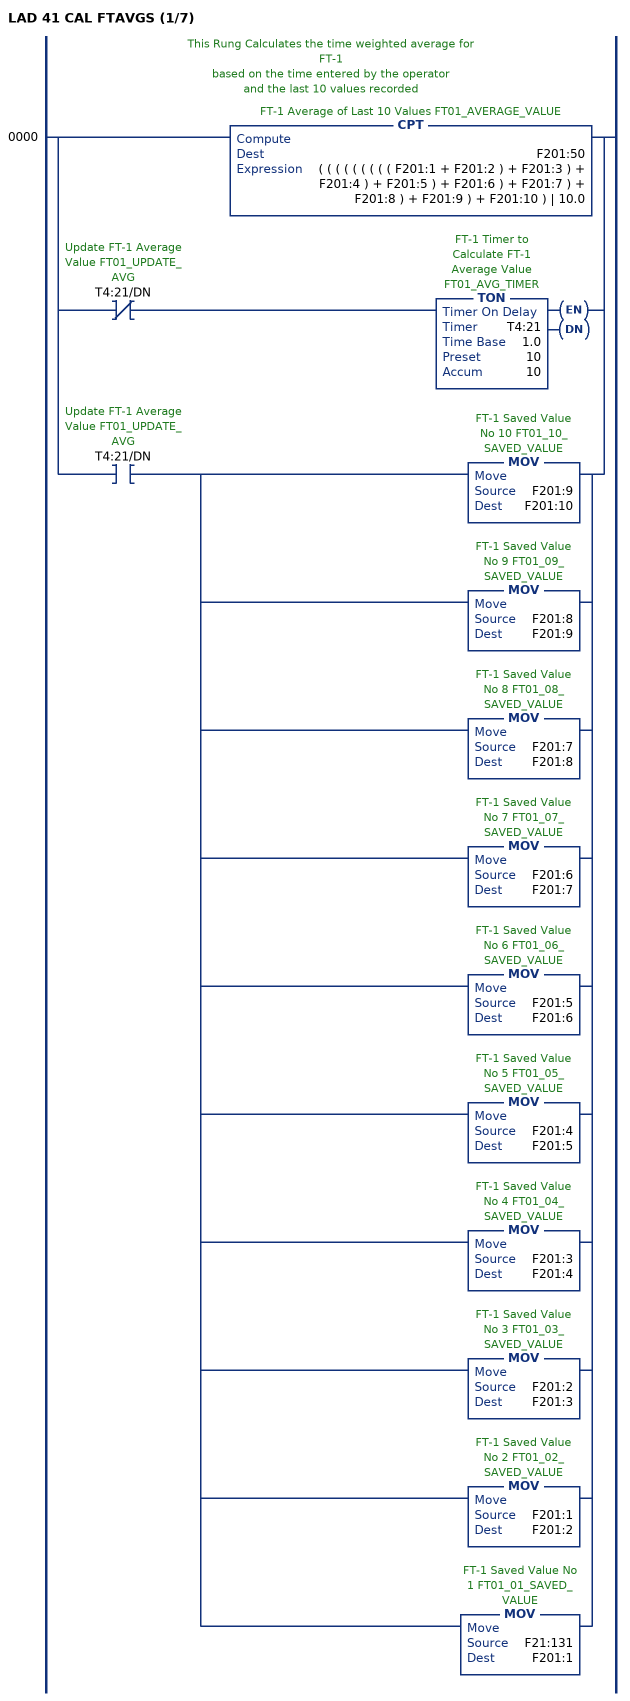
% Rung: 0 %
% This Rung Calculates the time weighted average for
% FT-1
% based on the time entered by the operator
% and the last 10 values recorded %
SOR BST CPT F201:50 " ( ( ( ( ( ( ( ( ( F201:1 + F201:2 ) + F201:3 ) + F201:4 ) + F201:5 ) + F201:6 ) + F201:7 ) + F201:8 ) + F201:9 ) + F201:10 ) | 10.0 " NXB XIO T4:21/DN TON T4:21 1.0 10 10 NXB XIC T4:21/DN BST MOV F201:9 F201:10 NXB MOV F201:8 F201:9 NXB MOV F201:7 F201:8 NXB MOV F201:6 F201:7 NXB MOV F201:5 F201:6 NXB MOV F201:4 F201:5 NXB MOV F201:3 F201:4 NXB MOV F201:2 F201:3 NXB MOV F201:1 F201:2 NXB MOV F21:131 F201:1 BND BND EOR
%   F201:50  FT01_AVERAGE_VALUE  "FT-1 Average of Last 10 Values" %
%   F201:1  FT01_01_SAVED_VALUE  "FT-1 Saved Value No 1" %
%   F201:2  FT01_02_SAVED_VALUE  "FT-1 Saved Value No 2" %
%   F201:3  FT01_03_SAVED_VALUE  "FT-1 Saved Value No 3" %
%   F201:4  FT01_04_SAVED_VALUE  "FT-1 Saved Value No 4" %
%   F201:5  FT01_05_SAVED_VALUE  "FT-1 Saved Value No 5" %
%   F201:6  FT01_06_SAVED_VALUE  "FT-1 Saved Value No 6" %
%   F201:7  FT01_07_SAVED_VALUE  "FT-1 Saved Value No 7" %
%   F201:8  FT01_08_SAVED_VALUE  "FT-1 Saved Value No 8" %
%   F201:9  FT01_09_SAVED_VALUE  "FT-1 Saved Value No 9" %
%   F201:10  FT01_10_SAVED_VALUE  "FT-1 Saved Value No 10" %
%   T4:21/DN  FT01_UPDATE_AVG  "Update FT-1 Average Value" %
%   T4:21  FT01_AVG_TIMER  "FT-1 Timer to Calculate FT-1 Average Value" %
%   F21:131  FT01  "FT-1 Flow Transmitter No-1" %

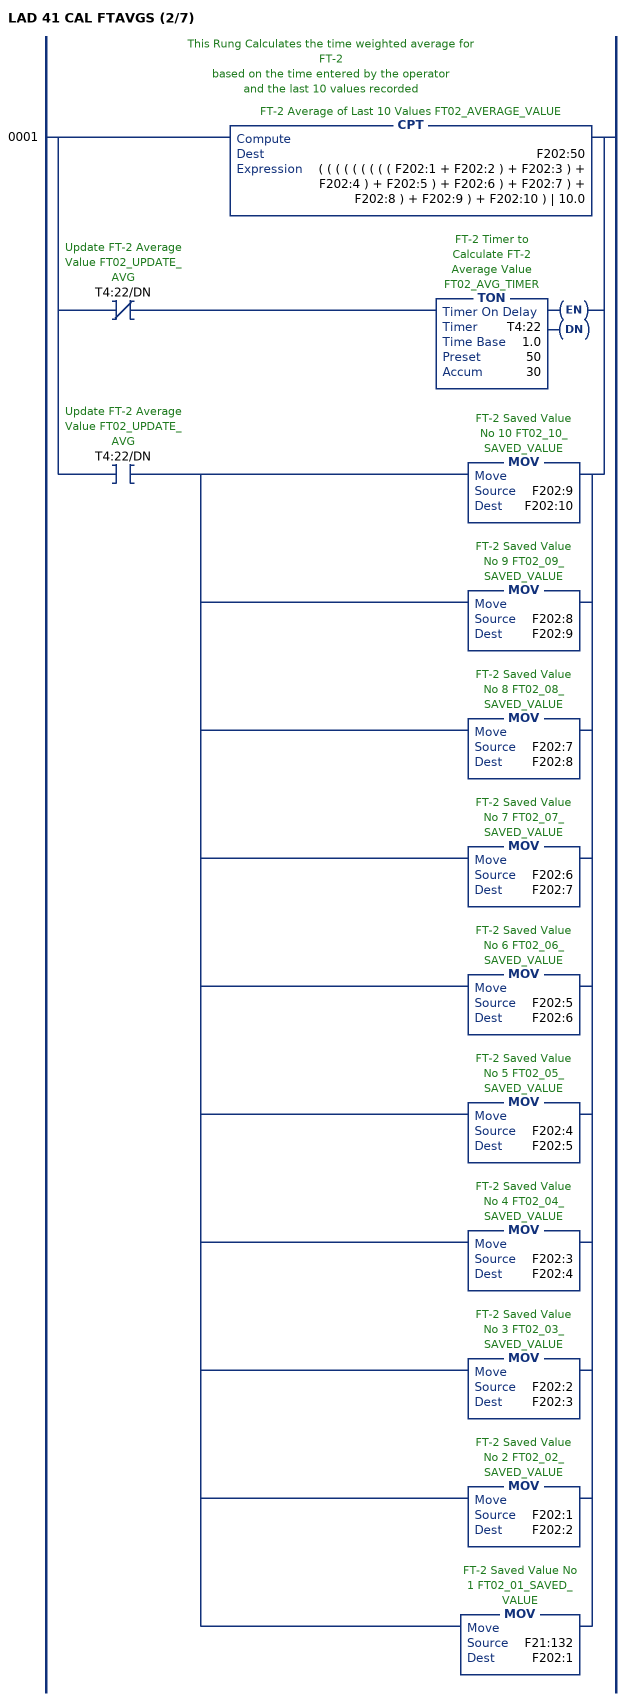
% Rung: 1 %
% This Rung Calculates the time weighted average for
% FT-2
% based on the time entered by the operator
% and the last 10 values recorded %
SOR BST CPT F202:50 " ( ( ( ( ( ( ( ( ( F202:1 + F202:2 ) + F202:3 ) + F202:4 ) + F202:5 ) + F202:6 ) + F202:7 ) + F202:8 ) + F202:9 ) + F202:10 ) | 10.0 " NXB XIO T4:22/DN TON T4:22 1.0 50 30 NXB XIC T4:22/DN BST MOV F202:9 F202:10 NXB MOV F202:8 F202:9 NXB MOV F202:7 F202:8 NXB MOV F202:6 F202:7 NXB MOV F202:5 F202:6 NXB MOV F202:4 F202:5 NXB MOV F202:3 F202:4 NXB MOV F202:2 F202:3 NXB MOV F202:1 F202:2 NXB MOV F21:132 F202:1 BND BND EOR
%   F202:50  FT02_AVERAGE_VALUE  "FT-2 Average of Last 10 Values" %
%   F202:1  FT02_01_SAVED_VALUE  "FT-2 Saved Value No 1" %
%   F202:2  FT02_02_SAVED_VALUE  "FT-2 Saved Value No 2" %
%   F202:3  FT02_03_SAVED_VALUE  "FT-2 Saved Value No 3" %
%   F202:4  FT02_04_SAVED_VALUE  "FT-2 Saved Value No 4" %
%   F202:5  FT02_05_SAVED_VALUE  "FT-2 Saved Value No 5" %
%   F202:6  FT02_06_SAVED_VALUE  "FT-2 Saved Value No 6" %
%   F202:7  FT02_07_SAVED_VALUE  "FT-2 Saved Value No 7" %
%   F202:8  FT02_08_SAVED_VALUE  "FT-2 Saved Value No 8" %
%   F202:9  FT02_09_SAVED_VALUE  "FT-2 Saved Value No 9" %
%   F202:10  FT02_10_SAVED_VALUE  "FT-2 Saved Value No 10" %
%   T4:22/DN  FT02_UPDATE_AVG  "Update FT-2 Average Value" %
%   T4:22  FT02_AVG_TIMER  "FT-2 Timer to Calculate FT-2 Average Value" %
%   F21:132  FT02  "FT-2 Flow Transmitter No-2" %

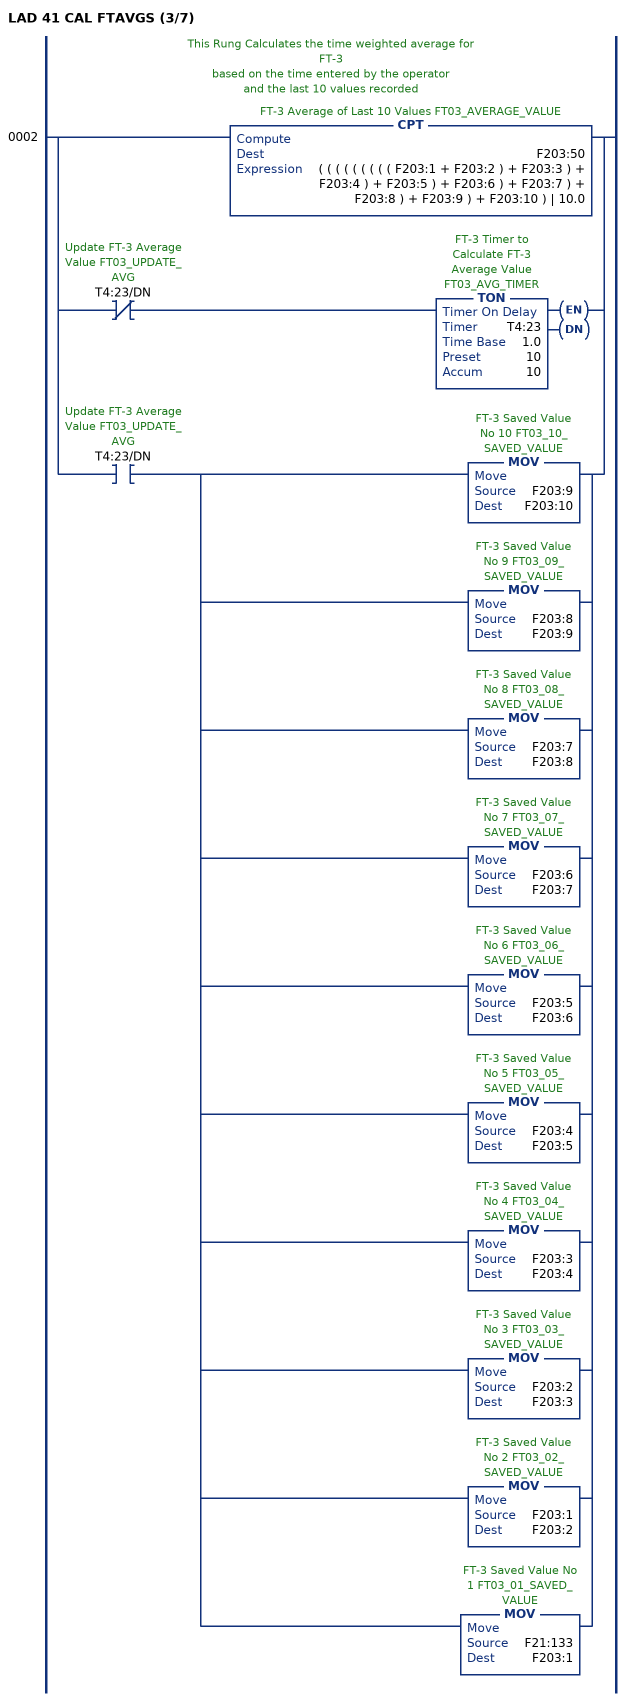
% Rung: 2 %
% This Rung Calculates the time weighted average for
% FT-3
% based on the time entered by the operator
% and the last 10 values recorded %
SOR BST CPT F203:50 " ( ( ( ( ( ( ( ( ( F203:1 + F203:2 ) + F203:3 ) + F203:4 ) + F203:5 ) + F203:6 ) + F203:7 ) + F203:8 ) + F203:9 ) + F203:10 ) | 10.0 " NXB XIO T4:23/DN TON T4:23 1.0 10 10 NXB XIC T4:23/DN BST MOV F203:9 F203:10 NXB MOV F203:8 F203:9 NXB MOV F203:7 F203:8 NXB MOV F203:6 F203:7 NXB MOV F203:5 F203:6 NXB MOV F203:4 F203:5 NXB MOV F203:3 F203:4 NXB MOV F203:2 F203:3 NXB MOV F203:1 F203:2 NXB MOV F21:133 F203:1 BND BND EOR
%   F203:50  FT03_AVERAGE_VALUE  "FT-3 Average of Last 10 Values" %
%   F203:1  FT03_01_SAVED_VALUE  "FT-3 Saved Value No 1" %
%   F203:2  FT03_02_SAVED_VALUE  "FT-3 Saved Value No 2" %
%   F203:3  FT03_03_SAVED_VALUE  "FT-3 Saved Value No 3" %
%   F203:4  FT03_04_SAVED_VALUE  "FT-3 Saved Value No 4" %
%   F203:5  FT03_05_SAVED_VALUE  "FT-3 Saved Value No 5" %
%   F203:6  FT03_06_SAVED_VALUE  "FT-3 Saved Value No 6" %
%   F203:7  FT03_07_SAVED_VALUE  "FT-3 Saved Value No 7" %
%   F203:8  FT03_08_SAVED_VALUE  "FT-3 Saved Value No 8" %
%   F203:9  FT03_09_SAVED_VALUE  "FT-3 Saved Value No 9" %
%   F203:10  FT03_10_SAVED_VALUE  "FT-3 Saved Value No 10" %
%   T4:23/DN  FT03_UPDATE_AVG  "Update FT-3 Average Value" %
%   T4:23  FT03_AVG_TIMER  "FT-3 Timer to Calculate FT-3 Average Value" %
%   F21:133  FT03  "FT-3 Flow Transmitter No-3" %

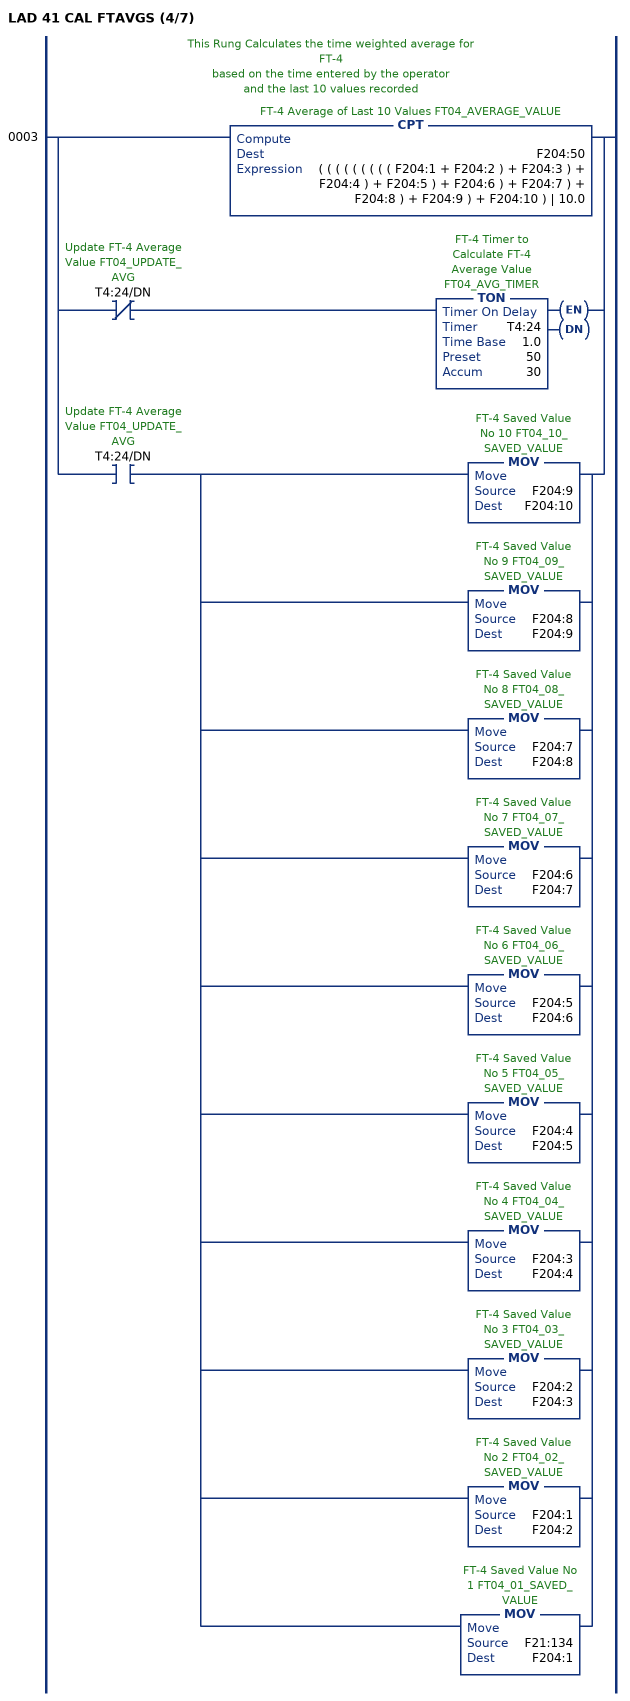
% Rung: 3 %
% This Rung Calculates the time weighted average for
% FT-4
% based on the time entered by the operator
% and the last 10 values recorded %
SOR BST CPT F204:50 " ( ( ( ( ( ( ( ( ( F204:1 + F204:2 ) + F204:3 ) + F204:4 ) + F204:5 ) + F204:6 ) + F204:7 ) + F204:8 ) + F204:9 ) + F204:10 ) | 10.0 " NXB XIO T4:24/DN TON T4:24 1.0 50 30 NXB XIC T4:24/DN BST MOV F204:9 F204:10 NXB MOV F204:8 F204:9 NXB MOV F204:7 F204:8 NXB MOV F204:6 F204:7 NXB MOV F204:5 F204:6 NXB MOV F204:4 F204:5 NXB MOV F204:3 F204:4 NXB MOV F204:2 F204:3 NXB MOV F204:1 F204:2 NXB MOV F21:134 F204:1 BND BND EOR
%   F204:50  FT04_AVERAGE_VALUE  "FT-4 Average of Last 10 Values" %
%   F204:1  FT04_01_SAVED_VALUE  "FT-4 Saved Value No 1" %
%   F204:2  FT04_02_SAVED_VALUE  "FT-4 Saved Value No 2" %
%   F204:3  FT04_03_SAVED_VALUE  "FT-4 Saved Value No 3" %
%   F204:4  FT04_04_SAVED_VALUE  "FT-4 Saved Value No 4" %
%   F204:5  FT04_05_SAVED_VALUE  "FT-4 Saved Value No 5" %
%   F204:6  FT04_06_SAVED_VALUE  "FT-4 Saved Value No 6" %
%   F204:7  FT04_07_SAVED_VALUE  "FT-4 Saved Value No 7" %
%   F204:8  FT04_08_SAVED_VALUE  "FT-4 Saved Value No 8" %
%   F204:9  FT04_09_SAVED_VALUE  "FT-4 Saved Value No 9" %
%   F204:10  FT04_10_SAVED_VALUE  "FT-4 Saved Value No 10" %
%   T4:24/DN  FT04_UPDATE_AVG  "Update FT-4 Average Value" %
%   T4:24  FT04_AVG_TIMER  "FT-4 Timer to Calculate FT-4 Average Value" %
%   F21:134  FT04  "FT-4 Flow Transmitter No-4" %

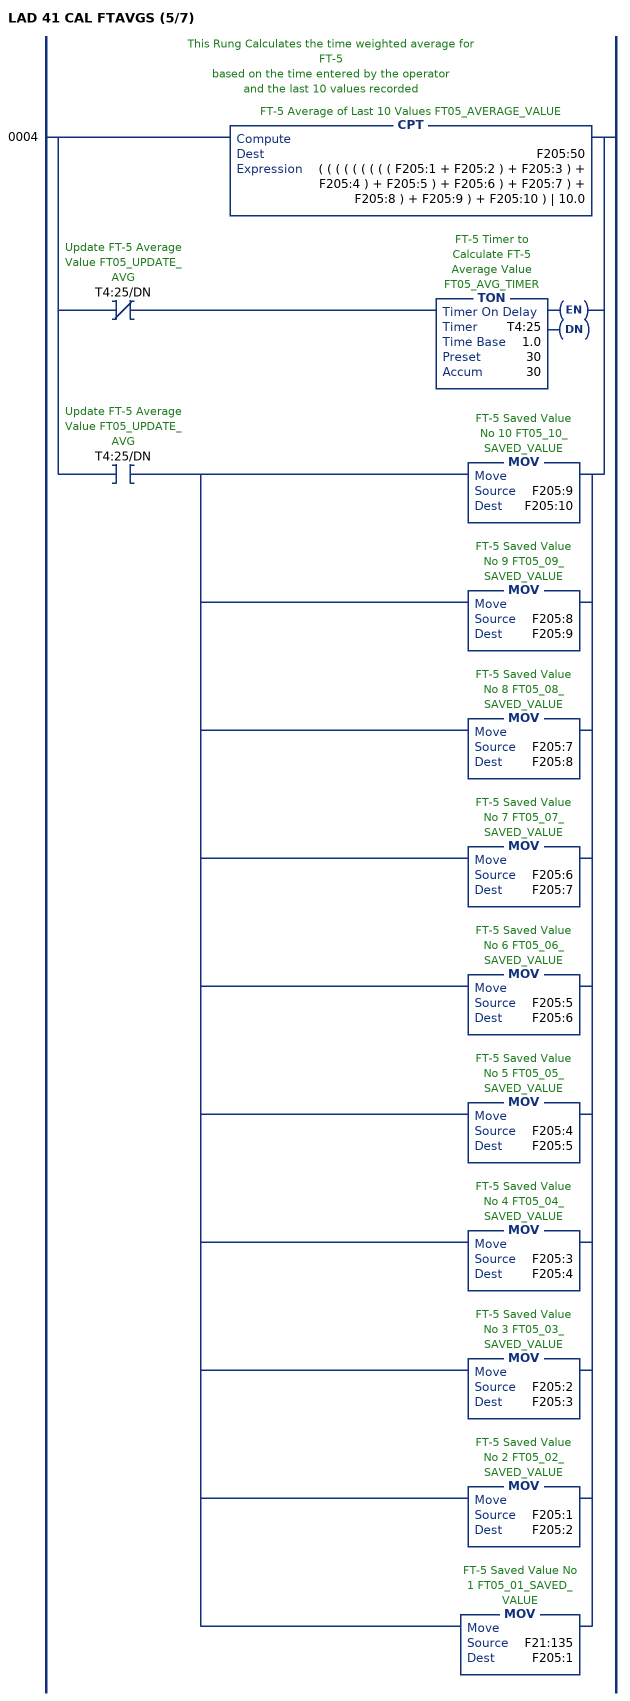
% Rung: 4 %
% This Rung Calculates the time weighted average for
% FT-5
% based on the time entered by the operator
% and the last 10 values recorded %
SOR BST CPT F205:50 " ( ( ( ( ( ( ( ( ( F205:1 + F205:2 ) + F205:3 ) + F205:4 ) + F205:5 ) + F205:6 ) + F205:7 ) + F205:8 ) + F205:9 ) + F205:10 ) | 10.0 " NXB XIO T4:25/DN TON T4:25 1.0 30 30 NXB XIC T4:25/DN BST MOV F205:9 F205:10 NXB MOV F205:8 F205:9 NXB MOV F205:7 F205:8 NXB MOV F205:6 F205:7 NXB MOV F205:5 F205:6 NXB MOV F205:4 F205:5 NXB MOV F205:3 F205:4 NXB MOV F205:2 F205:3 NXB MOV F205:1 F205:2 NXB MOV F21:135 F205:1 BND BND EOR
%   F205:50  FT05_AVERAGE_VALUE  "FT-5 Average of Last 10 Values" %
%   F205:1  FT05_01_SAVED_VALUE  "FT-5 Saved Value No 1" %
%   F205:2  FT05_02_SAVED_VALUE  "FT-5 Saved Value No 2" %
%   F205:3  FT05_03_SAVED_VALUE  "FT-5 Saved Value No 3" %
%   F205:4  FT05_04_SAVED_VALUE  "FT-5 Saved Value No 4" %
%   F205:5  FT05_05_SAVED_VALUE  "FT-5 Saved Value No 5" %
%   F205:6  FT05_06_SAVED_VALUE  "FT-5 Saved Value No 6" %
%   F205:7  FT05_07_SAVED_VALUE  "FT-5 Saved Value No 7" %
%   F205:8  FT05_08_SAVED_VALUE  "FT-5 Saved Value No 8" %
%   F205:9  FT05_09_SAVED_VALUE  "FT-5 Saved Value No 9" %
%   F205:10  FT05_10_SAVED_VALUE  "FT-5 Saved Value No 10" %
%   T4:25/DN  FT05_UPDATE_AVG  "Update FT-5 Average Value" %
%   T4:25  FT05_AVG_TIMER  "FT-5 Timer to Calculate FT-5 Average Value" %
%   F21:135  FT05  "FT-5 Flow Transmitter No-5" %

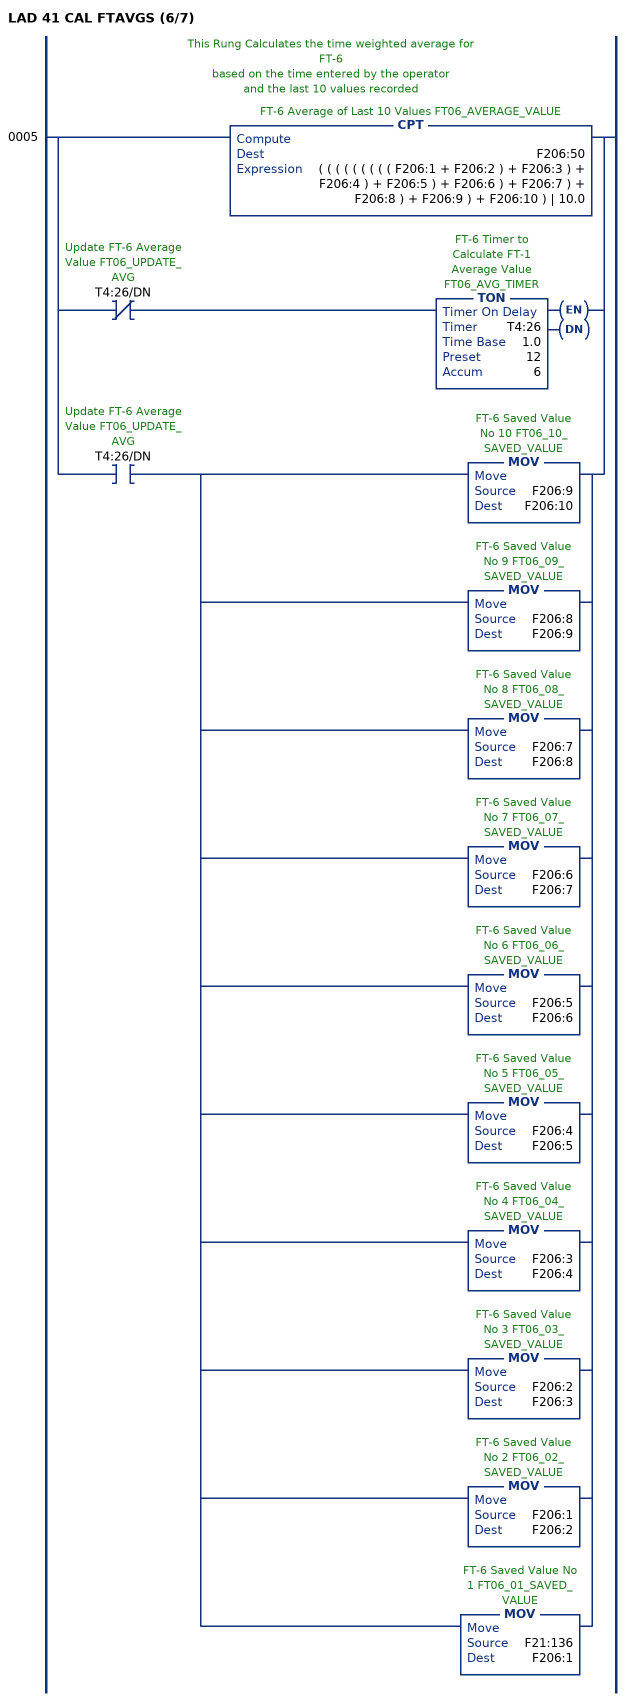
% Rung: 5 %
% This Rung Calculates the time weighted average for
% FT-6
% based on the time entered by the operator
% and the last 10 values recorded %
SOR BST CPT F206:50 " ( ( ( ( ( ( ( ( ( F206:1 + F206:2 ) + F206:3 ) + F206:4 ) + F206:5 ) + F206:6 ) + F206:7 ) + F206:8 ) + F206:9 ) + F206:10 ) | 10.0 " NXB XIO T4:26/DN TON T4:26 1.0 12 6 NXB XIC T4:26/DN BST MOV F206:9 F206:10 NXB MOV F206:8 F206:9 NXB MOV F206:7 F206:8 NXB MOV F206:6 F206:7 NXB MOV F206:5 F206:6 NXB MOV F206:4 F206:5 NXB MOV F206:3 F206:4 NXB MOV F206:2 F206:3 NXB MOV F206:1 F206:2 NXB MOV F21:136 F206:1 BND BND EOR
%   F206:50  FT06_AVERAGE_VALUE  "FT-6 Average of Last 10 Values" %
%   F206:1  FT06_01_SAVED_VALUE  "FT-6 Saved Value No 1" %
%   F206:2  FT06_02_SAVED_VALUE  "FT-6 Saved Value No 2" %
%   F206:3  FT06_03_SAVED_VALUE  "FT-6 Saved Value No 3" %
%   F206:4  FT06_04_SAVED_VALUE  "FT-6 Saved Value No 4" %
%   F206:5  FT06_05_SAVED_VALUE  "FT-6 Saved Value No 5" %
%   F206:6  FT06_06_SAVED_VALUE  "FT-6 Saved Value No 6" %
%   F206:7  FT06_07_SAVED_VALUE  "FT-6 Saved Value No 7" %
%   F206:8  FT06_08_SAVED_VALUE  "FT-6 Saved Value No 8" %
%   F206:9  FT06_09_SAVED_VALUE  "FT-6 Saved Value No 9" %
%   F206:10  FT06_10_SAVED_VALUE  "FT-6 Saved Value No 10" %
%   T4:26/DN  FT06_UPDATE_AVG  "Update FT-6 Average Value" %
%   T4:26  FT06_AVG_TIMER  "FT-6 Timer to Calculate FT-1 Average Value" %
%   F21:136  FT06  "FT-6 Flow Transmitter No-6" %

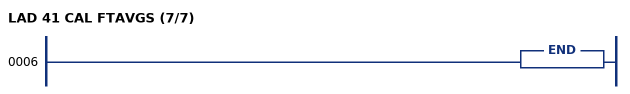
% Rung: 6 %
SOR END EOR

LADDER 42 "CALC LITS"    % Calculate LIT values %
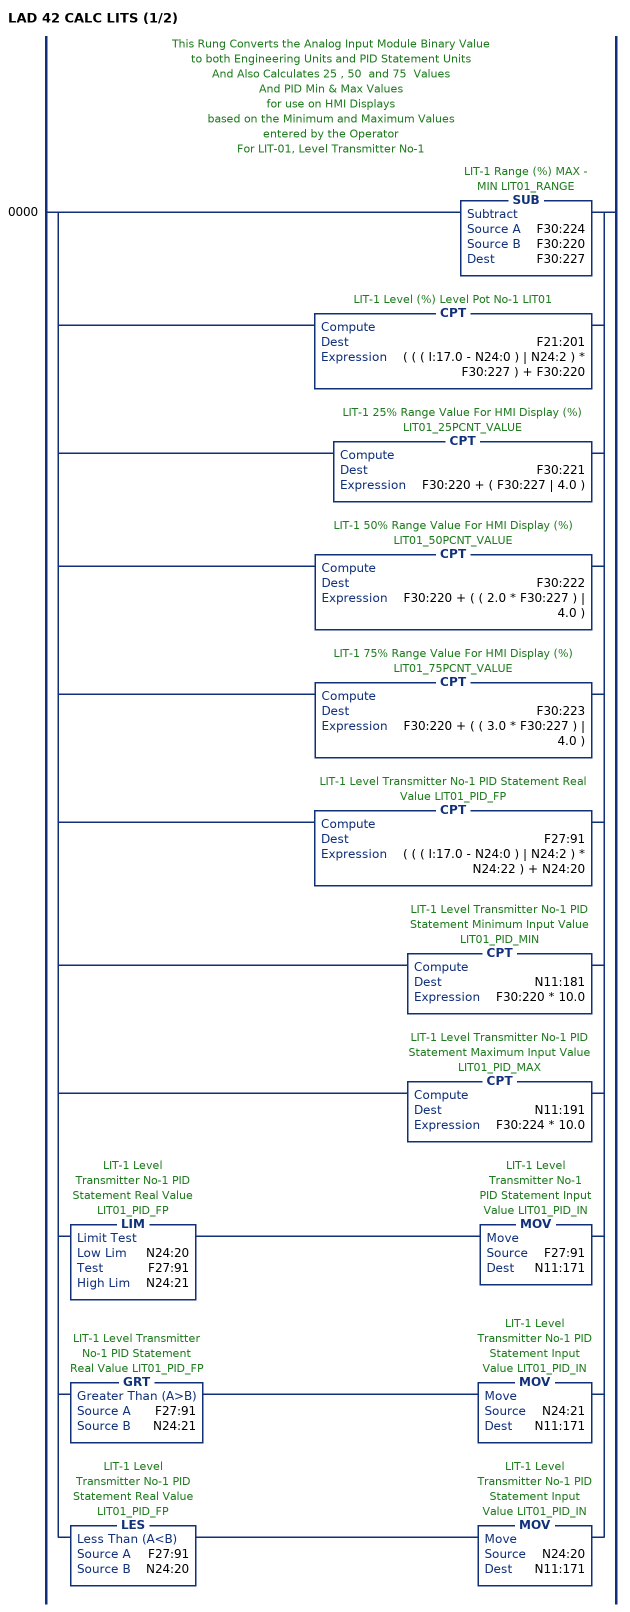
% Rung: 0 %
% This Rung Converts the Analog Input Module Binary Value
% to both Engineering Units and PID Statement Units
% And Also Calculates 25 , 50  and 75  Values
% And PID Min & Max Values
% for use on HMI Displays
% based on the Minimum and Maximum Values
% entered by the Operator
%    For LIT-01, Level Transmitter No-1 %
SOR BST SUB F30:224 F30:220 F30:227 NXB CPT F21:201 " ( ( ( I:17.0 - N24:0 ) | N24:2 ) * F30:227 ) + F30:220 " NXB CPT F30:221 " F30:220 + ( F30:227 | 4.0 ) " NXB CPT F30:222 " F30:220 + ( ( 2.0 * F30:227 ) | 4.0 ) " NXB CPT F30:223 " F30:220 + ( ( 3.0 * F30:227 ) | 4.0 ) " NXB CPT F27:91 " ( ( ( I:17.0 - N24:0 ) | N24:2 ) * N24:22 ) + N24:20 " NXB CPT N11:181 " F30:220 * 10.0 " NXB CPT N11:191 " F30:224 * 10.0 " NXB LIM N24:20 F27:91 N24:21 MOV F27:91 N11:171 NXB GRT F27:91 N24:21 MOV N24:21 N11:171 NXB LES F27:91 N24:20 MOV N24:20 N11:171 BND EOR
%   F30:224  LIT01_MAX  "LIT-1 Maximum Value (%)" %
%   F30:220  LIT01_MIN  "LIT-1 Minimum Value (%)" %
%   F30:227  LIT01_RANGE  "LIT-1 Range (%) MAX - MIN" %
%   F21:201  LIT01  "LIT-1 Level (%) Level Pot No-1" %
%   I:17.0  LIT01_BIN  "LIT-1 Binary Input From Transmitter Analog Input Module" %
%   N24:0  AI_CURRENT_MIN  "Analog Input Minimum Value = 4 mA DC (From AI Module)" %
%   N24:2  AI_CURRENT_RANGE  "Analog Input Current Range Value = (AI_MAX - AI_MIN) For Use Elswhere" %
%   F30:221  LIT01_25PCNT_VALUE  "LIT-1 25% Range Value For HMI Display (%)" %
%   F30:222  LIT01_50PCNT_VALUE  "LIT-1 50% Range Value For HMI Display (%)" %
%   F30:223  LIT01_75PCNT_VALUE  "LIT-1 75% Range Value For HMI Display (%)" %
%   F27:91  LIT01_PID_FP  "LIT-1 Level Transmitter No-1 PID Statement Real Value" %
%   N24:22  PID_RANGE  "PID Statement Range Value = (PID_MAX - PID_MIN) For Use Elswhere" %
%   N24:20  PID_MIN  "PID Statement Minimum Value" %
%   N11:181  LIT01_PID_MIN  "LIT-1 Level Transmitter No-1 PID Statement Minimum Input Value" %
%   N11:191  LIT01_PID_MAX  "LIT-1 Level Transmitter No-1 PID Statement Maximum Input Value" %
%   N24:21  PID_MAX  "PID Statement Maximum Value" %
%   N11:171  LIT01_PID_IN  "LIT-1 Level Transmitter No-1 PID Statement Input Value" %

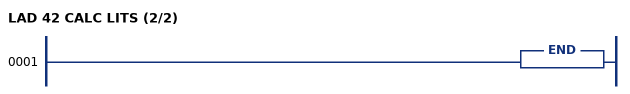
% Rung: 1 %
SOR END EOR

LADDER 43 "CALLC TITS"    % Calculate TITs %
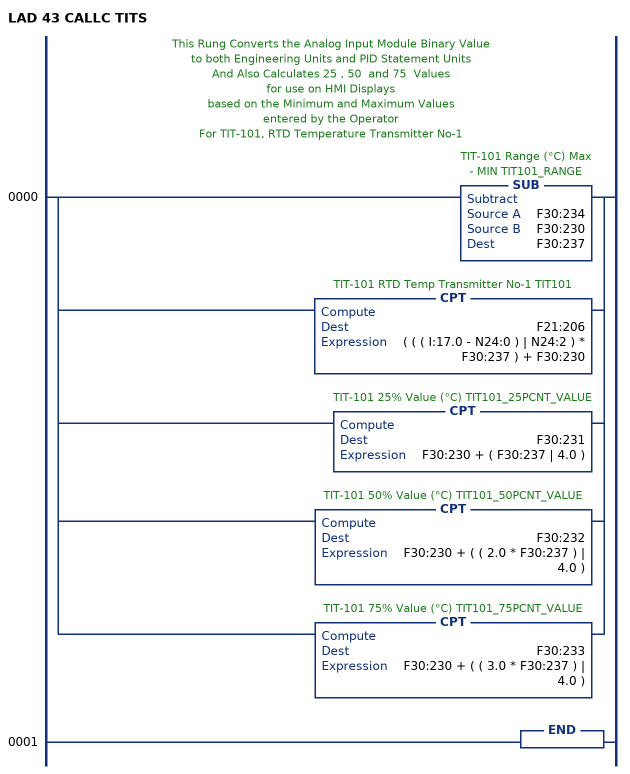
% Rung: 0 %
% This Rung Converts the Analog Input Module Binary Value
% to both Engineering Units and PID Statement Units
% And Also Calculates 25 , 50  and 75  Values
% 
% for use on HMI Displays
% based on the Minimum and Maximum Values
% entered by the Operator
%    For TIT-101, RTD Temperature Transmitter No-1 %
SOR BST SUB F30:234 F30:230 F30:237 NXB CPT F21:206 " ( ( ( I:17.0 - N24:0 ) | N24:2 ) * F30:237 ) + F30:230 " NXB CPT F30:231 " F30:230 + ( F30:237 | 4.0 ) " NXB CPT F30:232 " F30:230 + ( ( 2.0 * F30:237 ) | 4.0 ) " NXB CPT F30:233 " F30:230 + ( ( 3.0 * F30:237 ) | 4.0 ) " BND EOR
%   F30:234  TIT101_MAX  "TIT-101 Maximum Value (°C)" %
%   F30:230  TIT101_MIN  "TIT-101 Minimum Value (°C)" %
%   F30:237  TIT101_RANGE  "TIT-101 Range (°C) Max - MIN" %
%   F21:206  TIT101  "TIT-101 RTD Temp Transmitter No-1" %
%   I:17.0  LIT01_BIN  "LIT-1 Binary Input From Transmitter Analog Input Module" %
%   N24:0  AI_CURRENT_MIN  "Analog Input Minimum Value = 4 mA DC (From AI Module)" %
%   N24:2  AI_CURRENT_RANGE  "Analog Input Current Range Value = (AI_MAX - AI_MIN) For Use Elswhere" %
%   F30:231  TIT101_25PCNT_VALUE  "TIT-101 25% Value (°C)" %
%   F30:232  TIT101_50PCNT_VALUE  "TIT-101 50% Value (°C)" %
%   F30:233  TIT101_75PCNT_VALUE  "TIT-101 75% Value (°C)" %
% Rung: 1 %
SOR END EOR

LADDER 48 "EF-1"    % Process Area Exhaust Fan Controls %
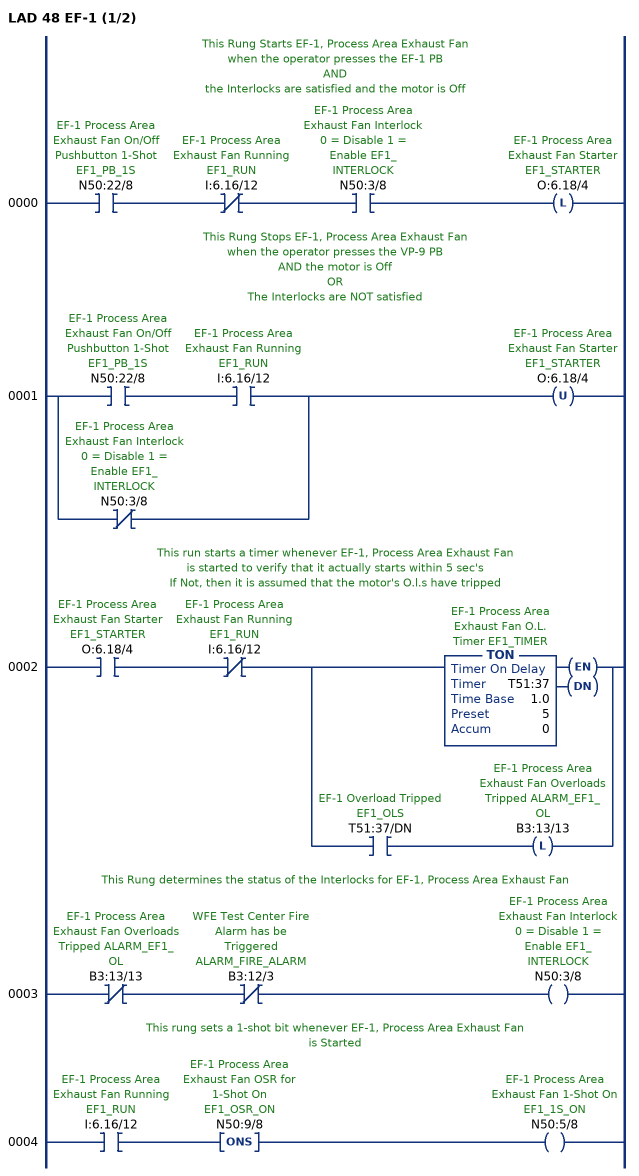
% Rung: 0 %
% This Rung Starts EF-1, Process Area Exhaust Fan
% when the operator presses the EF-1 PB
% AND
% the Interlocks are satisfied and the motor is Off %
SOR XIC N50:22/8 XIO I:6.16/12 XIC N50:3/8 OTL O:6.18/4 EOR
%   N50:22/8  EF1_PB_1S  "EF-1 Process Area Exhaust Fan On/Off Pushbutton 1-Shot" %
%   I:6.16/12  EF1_RUN  "EF-1 Process Area Exhaust Fan Running" %
%   N50:3/8  EF1_INTERLOCK  "EF-1 Process Area Exhaust Fan Interlock 0 = Disable 1 = Enable" %
%   O:6.18/4  EF1_STARTER  "EF-1 Process Area Exhaust Fan Starter" %
% Rung: 1 %
% This Rung Stops EF-1, Process Area Exhaust Fan
% when the operator presses the VP-9 PB
% AND the motor is Off
% OR
% The Interlocks are NOT satisfied %
SOR BST XIC N50:22/8 XIC I:6.16/12 NXB XIO N50:3/8 BND OTU O:6.18/4 EOR
%   N50:22/8  EF1_PB_1S  "EF-1 Process Area Exhaust Fan On/Off Pushbutton 1-Shot" %
%   I:6.16/12  EF1_RUN  "EF-1 Process Area Exhaust Fan Running" %
%   N50:3/8  EF1_INTERLOCK  "EF-1 Process Area Exhaust Fan Interlock 0 = Disable 1 = Enable" %
%   O:6.18/4  EF1_STARTER  "EF-1 Process Area Exhaust Fan Starter" %
% Rung: 2 %
% This run starts a timer whenever EF-1, Process Area Exhaust Fan
% is started to verify that it actually starts within 5 sec's
% If Not, then it is assumed that the motor's O.l.s have tripped %
SOR XIC O:6.18/4 XIO I:6.16/12 BST TON T51:37 1.0 5 0 NXB XIC T51:37/DN OTL B3:13/13 BND EOR
%   O:6.18/4  EF1_STARTER  "EF-1 Process Area Exhaust Fan Starter" %
%   I:6.16/12  EF1_RUN  "EF-1 Process Area Exhaust Fan Running" %
%   T51:37  EF1_TIMER  "EF-1 Process Area Exhaust Fan O.L. Timer" %
%   T51:37/DN  EF1_OLS  "EF-1 Overload Tripped" %
%   B3:13/13  ALARM_EF1_OL  "EF-1 Process Area Exhaust Fan Overloads Tripped" %
% Rung: 3 %
% This Rung determines the status of the Interlocks for EF-1, Process Area Exhaust Fan %
SOR XIO B3:13/13 XIO B3:12/3 OTE N50:3/8 EOR
%   B3:13/13  ALARM_EF1_OL  "EF-1 Process Area Exhaust Fan Overloads Tripped" %
%   B3:12/3  ALARM_FIRE_ALARM  "WFE Test Center Fire Alarm has be Triggered" %
%   N50:3/8  EF1_INTERLOCK  "EF-1 Process Area Exhaust Fan Interlock 0 = Disable 1 = Enable" %
% Rung: 4 %
% This rung sets a 1-shot bit whenever EF-1, Process Area Exhaust Fan
% is Started %
SOR XIC I:6.16/12 OSR N50:9/8 OTE N50:5/8 EOR
%   I:6.16/12  EF1_RUN  "EF-1 Process Area Exhaust Fan Running" %
%   N50:9/8  EF1_OSR_ON  "EF-1 Process Area Exhaust Fan OSR for 1-Shot On" %
%   N50:5/8  EF1_1S_ON  "EF-1 Process Area Exhaust Fan 1-Shot On" %

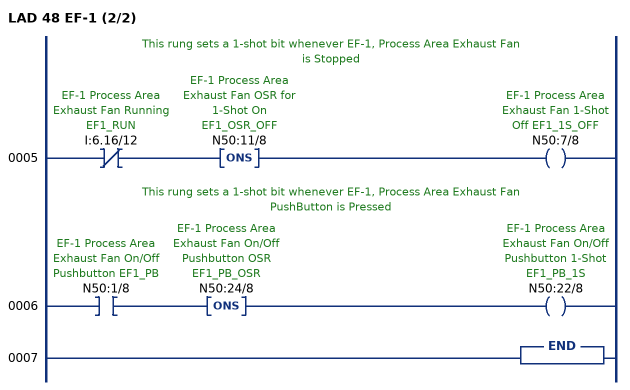
% Rung: 5 %
% This rung sets a 1-shot bit whenever EF-1, Process Area Exhaust Fan
% is Stopped %
SOR XIO I:6.16/12 OSR N50:11/8 OTE N50:7/8 EOR
%   I:6.16/12  EF1_RUN  "EF-1 Process Area Exhaust Fan Running" %
%   N50:11/8  EF1_OSR_OFF  "EF-1 Process Area Exhaust Fan OSR for 1-Shot On" %
%   N50:7/8  EF1_1S_OFF  "EF-1 Process Area Exhaust Fan 1-Shot Off" %
% Rung: 6 %
% This rung sets a 1-shot bit whenever EF-1, Process Area Exhaust Fan
% PushButton is Pressed %
SOR XIC N50:1/8 OSR N50:24/8 OTE N50:22/8 EOR
%   N50:1/8  EF1_PB  "EF-1 Process Area Exhaust Fan On/Off Pushbutton" %
%   N50:24/8  EF1_PB_OSR  "EF-1 Process Area Exhaust Fan On/Off Pushbutton OSR" %
%   N50:22/8  EF1_PB_1S  "EF-1 Process Area Exhaust Fan On/Off Pushbutton 1-Shot" %
% Rung: 7 %
SOR END EOR

LADDER 49 "EF-2"    % Utility Room Exhaust Fan Controls %
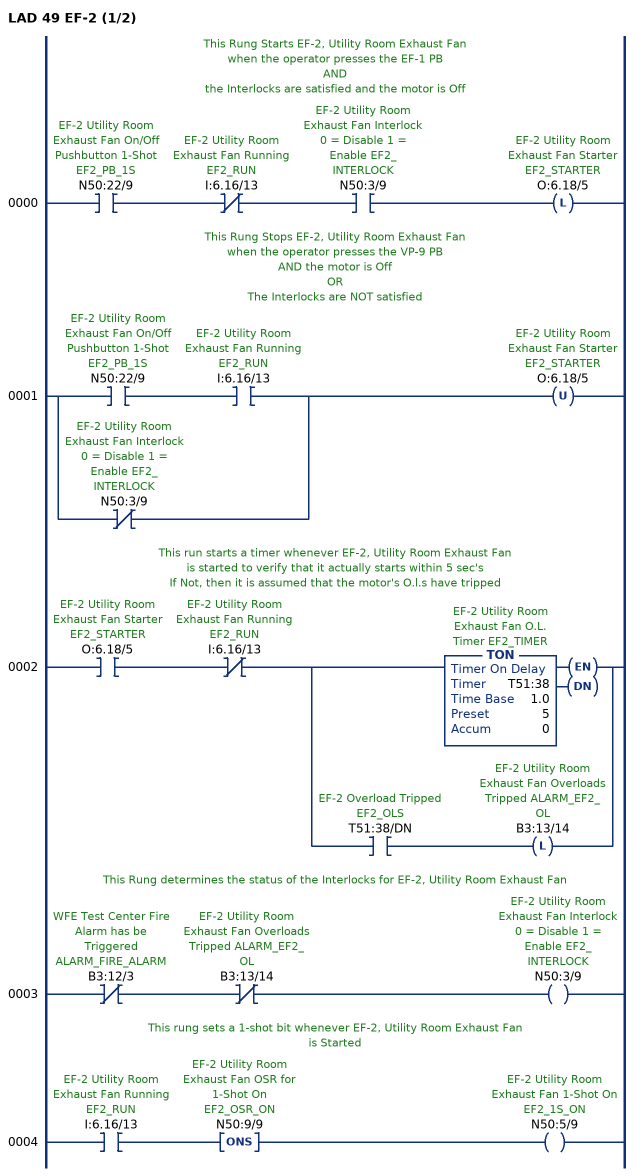
% Rung: 0 %
% This Rung Starts EF-2, Utility Room Exhaust Fan
% when the operator presses the EF-1 PB
% AND
% the Interlocks are satisfied and the motor is Off %
SOR XIC N50:22/9 XIO I:6.16/13 XIC N50:3/9 OTL O:6.18/5 EOR
%   N50:22/9  EF2_PB_1S  "EF-2 Utility Room Exhaust Fan On/Off Pushbutton 1-Shot" %
%   I:6.16/13  EF2_RUN  "EF-2 Utility Room Exhaust Fan Running" %
%   N50:3/9  EF2_INTERLOCK  "EF-2 Utility Room Exhaust Fan Interlock 0 = Disable 1 = Enable" %
%   O:6.18/5  EF2_STARTER  "EF-2 Utility Room Exhaust Fan Starter" %
% Rung: 1 %
% This Rung Stops EF-2, Utility Room Exhaust Fan
% when the operator presses the VP-9 PB
% AND the motor is Off
% OR
% The Interlocks are NOT satisfied %
SOR BST XIC N50:22/9 XIC I:6.16/13 NXB XIO N50:3/9 BND OTU O:6.18/5 EOR
%   N50:22/9  EF2_PB_1S  "EF-2 Utility Room Exhaust Fan On/Off Pushbutton 1-Shot" %
%   I:6.16/13  EF2_RUN  "EF-2 Utility Room Exhaust Fan Running" %
%   N50:3/9  EF2_INTERLOCK  "EF-2 Utility Room Exhaust Fan Interlock 0 = Disable 1 = Enable" %
%   O:6.18/5  EF2_STARTER  "EF-2 Utility Room Exhaust Fan Starter" %
% Rung: 2 %
% This run starts a timer whenever EF-2, Utility Room Exhaust Fan
% is started to verify that it actually starts within 5 sec's
% If Not, then it is assumed that the motor's O.l.s have tripped %
SOR XIC O:6.18/5 XIO I:6.16/13 BST TON T51:38 1.0 5 0 NXB XIC T51:38/DN OTL B3:13/14 BND EOR
%   O:6.18/5  EF2_STARTER  "EF-2 Utility Room Exhaust Fan Starter" %
%   I:6.16/13  EF2_RUN  "EF-2 Utility Room Exhaust Fan Running" %
%   T51:38  EF2_TIMER  "EF-2 Utility Room Exhaust Fan O.L. Timer" %
%   T51:38/DN  EF2_OLS  "EF-2 Overload Tripped" %
%   B3:13/14  ALARM_EF2_OL  "EF-2 Utility Room Exhaust Fan Overloads Tripped" %
% Rung: 3 %
% This Rung determines the status of the Interlocks for EF-2, Utility Room Exhaust Fan %
SOR XIO B3:12/3 XIO B3:13/14 OTE N50:3/9 EOR
%   B3:12/3  ALARM_FIRE_ALARM  "WFE Test Center Fire Alarm has be Triggered" %
%   B3:13/14  ALARM_EF2_OL  "EF-2 Utility Room Exhaust Fan Overloads Tripped" %
%   N50:3/9  EF2_INTERLOCK  "EF-2 Utility Room Exhaust Fan Interlock 0 = Disable 1 = Enable" %
% Rung: 4 %
% This rung sets a 1-shot bit whenever EF-2, Utility Room Exhaust Fan
% is Started %
SOR XIC I:6.16/13 OSR N50:9/9 OTE N50:5/9 EOR
%   I:6.16/13  EF2_RUN  "EF-2 Utility Room Exhaust Fan Running" %
%   N50:9/9  EF2_OSR_ON  "EF-2 Utility Room Exhaust Fan OSR for 1-Shot On" %
%   N50:5/9  EF2_1S_ON  "EF-2 Utility Room Exhaust Fan 1-Shot On" %

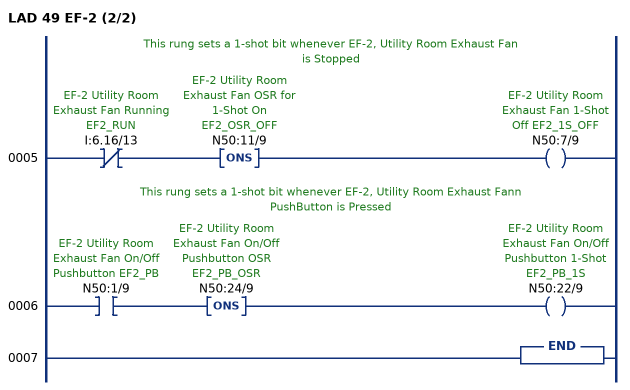
% Rung: 5 %
% This rung sets a 1-shot bit whenever EF-2, Utility Room Exhaust Fan
% is Stopped %
SOR XIO I:6.16/13 OSR N50:11/9 OTE N50:7/9 EOR
%   I:6.16/13  EF2_RUN  "EF-2 Utility Room Exhaust Fan Running" %
%   N50:11/9  EF2_OSR_OFF  "EF-2 Utility Room Exhaust Fan OSR for 1-Shot On" %
%   N50:7/9  EF2_1S_OFF  "EF-2 Utility Room Exhaust Fan 1-Shot Off" %
% Rung: 6 %
% This rung sets a 1-shot bit whenever EF-2, Utility Room Exhaust Fann
% PushButton is Pressed %
SOR XIC N50:1/9 OSR N50:24/9 OTE N50:22/9 EOR
%   N50:1/9  EF2_PB  "EF-2 Utility Room Exhaust Fan On/Off Pushbutton" %
%   N50:24/9  EF2_PB_OSR  "EF-2 Utility Room Exhaust Fan On/Off Pushbutton OSR" %
%   N50:22/9  EF2_PB_1S  "EF-2 Utility Room Exhaust Fan On/Off Pushbutton 1-Shot" %
% Rung: 7 %
SOR END EOR

LADDER 50 "EV-01"    % EV-1 Rotor Controls %
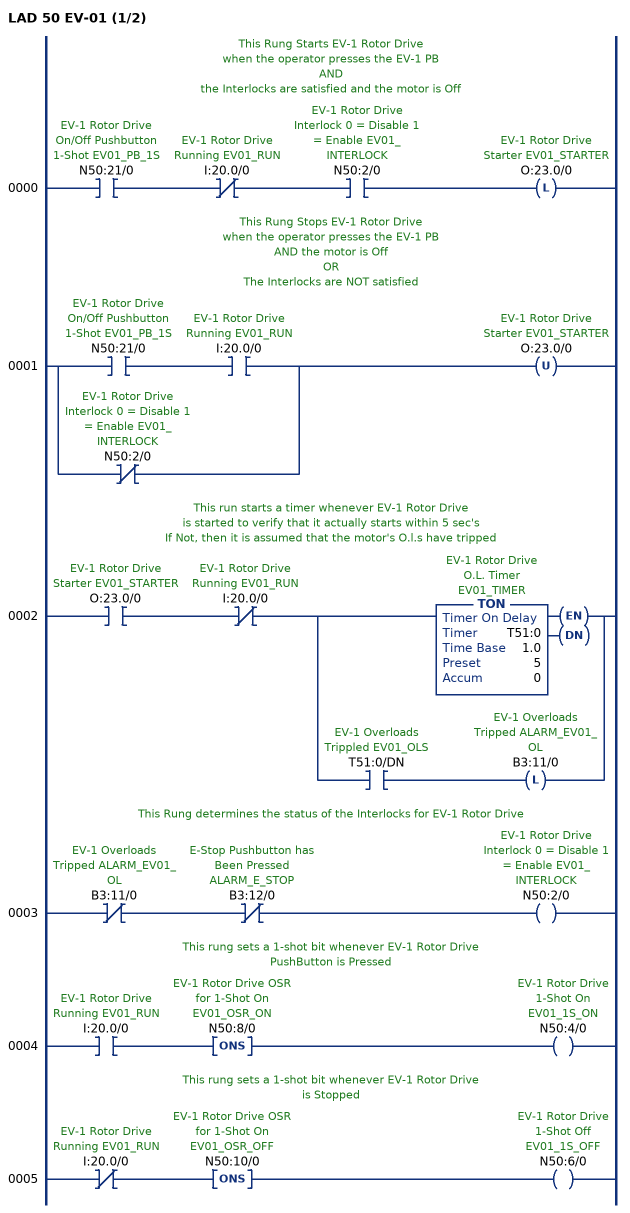
% Rung: 0 %
% This Rung Starts EV-1 Rotor Drive
% when the operator presses the EV-1 PB
% AND
% the Interlocks are satisfied and the motor is Off %
SOR XIC N50:21/0 XIO I:20.0/0 XIC N50:2/0 OTL O:23.0/0 EOR
%   N50:21/0  EV01_PB_1S  "EV-1 Rotor Drive On/Off Pushbutton 1-Shot" %
%   I:20.0/0  EV01_RUN  "EV-1 Rotor Drive Running" %
%   N50:2/0  EV01_INTERLOCK  "EV-1 Rotor Drive Interlock 0 = Disable 1 = Enable" %
%   O:23.0/0  EV01_STARTER  "EV-1 Rotor Drive Starter" %
% Rung: 1 %
% This Rung Stops EV-1 Rotor Drive
% when the operator presses the EV-1 PB
% AND the motor is Off
% OR
% The Interlocks are NOT satisfied %
SOR BST XIC N50:21/0 XIC I:20.0/0 NXB XIO N50:2/0 BND OTU O:23.0/0 EOR
%   N50:21/0  EV01_PB_1S  "EV-1 Rotor Drive On/Off Pushbutton 1-Shot" %
%   I:20.0/0  EV01_RUN  "EV-1 Rotor Drive Running" %
%   N50:2/0  EV01_INTERLOCK  "EV-1 Rotor Drive Interlock 0 = Disable 1 = Enable" %
%   O:23.0/0  EV01_STARTER  "EV-1 Rotor Drive Starter" %
% Rung: 2 %
% This run starts a timer whenever EV-1 Rotor Drive
% is started to verify that it actually starts within 5 sec's
% If Not, then it is assumed that the motor's O.l.s have tripped %
SOR XIC O:23.0/0 XIO I:20.0/0 BST TON T51:0 1.0 5 0 NXB XIC T51:0/DN OTL B3:11/0 BND EOR
%   O:23.0/0  EV01_STARTER  "EV-1 Rotor Drive Starter" %
%   I:20.0/0  EV01_RUN  "EV-1 Rotor Drive Running" %
%   T51:0  EV01_TIMER  "EV-1 Rotor Drive O.L. Timer" %
%   T51:0/DN  EV01_OLS  "EV-1 Overloads Trippled" %
%   B3:11/0  ALARM_EV01_OL  "EV-1 Overloads Tripped" %
% Rung: 3 %
% This Rung determines the status of the Interlocks for EV-1 Rotor Drive %
SOR XIO B3:11/0 XIO B3:12/0 OTE N50:2/0 EOR
%   B3:11/0  ALARM_EV01_OL  "EV-1 Overloads Tripped" %
%   B3:12/0  ALARM_E_STOP  "E-Stop Pushbutton has Been Pressed" %
%   N50:2/0  EV01_INTERLOCK  "EV-1 Rotor Drive Interlock 0 = Disable 1 = Enable" %
% Rung: 4 %
% This rung sets a 1-shot bit whenever EV-1 Rotor Drive
% PushButton is Pressed %
SOR XIC I:20.0/0 OSR N50:8/0 OTE N50:4/0 EOR
%   I:20.0/0  EV01_RUN  "EV-1 Rotor Drive Running" %
%   N50:8/0  EV01_OSR_ON  "EV-1 Rotor Drive OSR for 1-Shot On" %
%   N50:4/0  EV01_1S_ON  "EV-1 Rotor Drive 1-Shot On" %
% Rung: 5 %
% This rung sets a 1-shot bit whenever EV-1 Rotor Drive
% is Stopped %
SOR XIO I:20.0/0 OSR N50:10/0 OTE N50:6/0 EOR
%   I:20.0/0  EV01_RUN  "EV-1 Rotor Drive Running" %
%   N50:10/0  EV01_OSR_OFF  "EV-1 Rotor Drive OSR for 1-Shot On" %
%   N50:6/0  EV01_1S_OFF  "EV-1 Rotor Drive 1-Shot Off" %

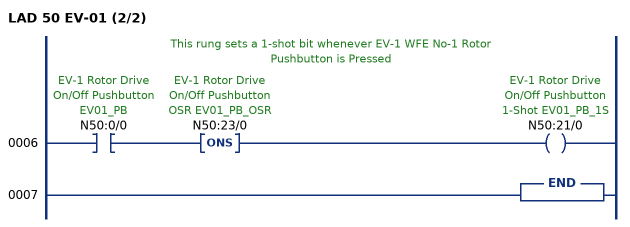
% Rung: 6 %
% This rung sets a 1-shot bit whenever EV-1 WFE No-1 Rotor
% Pushbutton is Pressed %
SOR XIC N50:0/0 OSR N50:23/0 OTE N50:21/0 EOR
%   N50:0/0  EV01_PB  "EV-1 Rotor Drive On/Off Pushbutton" %
%   N50:23/0  EV01_PB_OSR  "EV-1 Rotor Drive On/Off Pushbutton OSR" %
%   N50:21/0  EV01_PB_1S  "EV-1 Rotor Drive On/Off Pushbutton 1-Shot" %
% Rung: 7 %
SOR END EOR

LADDER 51 "EV-02"    % EV-2 Rotor Drive VFD Controls %
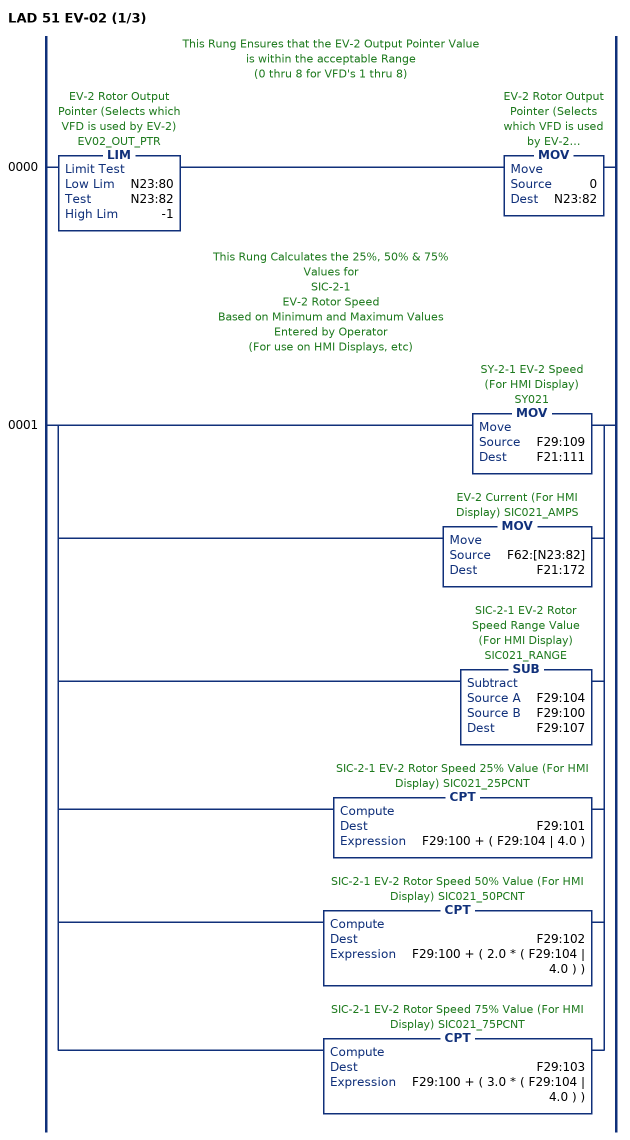
% Rung: 0 %
% This Rung Ensures that the EV-2 Output Pointer Value
% is within the acceptable Range
% (0 thru 8 for VFD's 1 thru 8) %
SOR LIM N23:80 N23:82 -1 MOV 0 N23:82 EOR
%   N23:80  MAX_VFD_ALLOWED_1  "Maximum Number of VFDs Available Plus 1" %
%   N23:82  EV02_OUT_PTR  "EV-2 Rotor Output Pointer (Selects which VFD is used by EV-2)" %
% Rung: 1 %
% This Rung Calculates the 25%, 50% & 75%
% Values for
% SIC-2-1
% EV-2 Rotor Speed
% Based on Minimum and Maximum Values
% Entered by Operator
% (For use on HMI Displays, etc) %
SOR BST MOV F29:109 F21:111 NXB MOV F62:[N23:82] F21:172 NXB SUB F29:104 F29:100 F29:107 NXB CPT F29:101 " F29:100 + ( F29:104 | 4.0 ) " NXB CPT F29:102 " F29:100 + ( 2.0 * ( F29:104 | 4.0 ) ) " NXB CPT F29:103 " F29:100 + ( 3.0 * ( F29:104 | 4.0 ) ) " BND EOR
%   F29:109  SIC021_SP_FP  "SIC-2-1 EV-2 Rotor Speed Setpoint Value (For HMI Display)" %
%   F21:111  SY021  "SY-2-1 EV-2 Speed (For HMI Display)" %
%   N23:82  EV02_OUT_PTR  "EV-2 Rotor Output Pointer (Selects which VFD is used by EV-2)" %
%   F21:172  SIC021_AMPS  "EV-2 Current (For HMI Display)" %
%   F29:104  SIC021_MAX  "SIC-2-1 EV-2 Rotor Speed 100% Value (For HMI Display)" %
%   F29:100  SIC021_MIN  "SIC-2-1 EV-2 Rotor Speed 0% Value (For HMI Display)" %
%   F29:107  SIC021_RANGE  "SIC-2-1 EV-2 Rotor Speed Range Value (For HMI Display)" %
%   F29:101  SIC021_25PCNT  "SIC-2-1 EV-2 Rotor Speed 25% Value (For HMI Display)" %
%   F29:102  SIC021_50PCNT  "SIC-2-1 EV-2 Rotor Speed 50% Value (For HMI Display)" %
%   F29:103  SIC021_75PCNT  "SIC-2-1 EV-2 Rotor Speed 75% Value (For HMI Display)" %

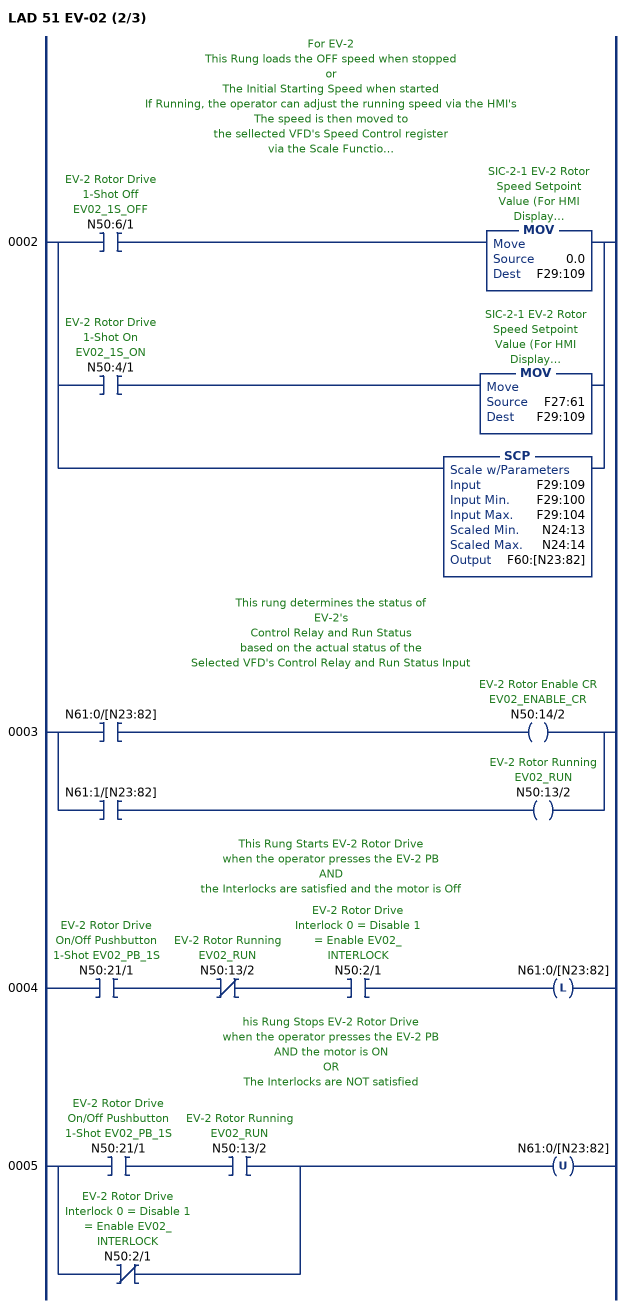
% Rung: 2 %
% For EV-2
% This Rung loads the OFF speed when stopped
% or
% The Initial Starting Speed when started
% If Running, the operator can adjust the running speed via the HMI's
% The speed is then moved to
% the sellected VFD's Speed Control register
% via the Scale Function
% to actually adjust the VFD's Speed %
SOR BST XIC N50:6/1 MOV 0.0 F29:109 NXB XIC N50:4/1 MOV F27:61 F29:109 NXB SCP F29:109 F29:100 F29:104 N24:13 N24:14 F60:[N23:82] BND EOR
%   N50:6/1  EV02_1S_OFF  "EV-2 Rotor Drive 1-Shot Off" %
%   F29:109  SIC021_SP_FP  "SIC-2-1 EV-2 Rotor Speed Setpoint Value (For HMI Display)" %
%   N50:4/1  EV02_1S_ON  "EV-2 Rotor Drive 1-Shot On" %
%   F27:61  SIC021_INIT_SP  "SY-2-1 Initial Speed Setpoint (RPM)" %
%   F29:100  SIC021_MIN  "SIC-2-1 EV-2 Rotor Speed 0% Value (For HMI Display)" %
%   F29:104  SIC021_MAX  "SIC-2-1 EV-2 Rotor Speed 100% Value (For HMI Display)" %
%   N24:13  AO_MIN_OE4  "Analog Output Minimum Value Generates 4 mA DC (To OE4 AO Module)" %
%   N24:14  AO_MAX_OE4  "Analog Output Maximum Value Generates 20 mA DC (To OE4 AO Module)" %
%   N23:82  EV02_OUT_PTR  "EV-2 Rotor Output Pointer (Selects which VFD is used by EV-2)" %
% Rung: 3 %
% This rung determines the status of
% EV-2's
% Control Relay and Run Status
% based on the actual status of the
% Selected VFD's Control Relay and Run Status Input %
SOR BST XIC N61:0/[N23:82] OTE N50:14/2 NXB XIC N61:1/[N23:82] OTE N50:13/2 BND EOR
%   N61:0  VFD_ENABLE_BITS  "These Bits Enable the appropriate VFD" %
%   N23:82  EV02_OUT_PTR  "EV-2 Rotor Output Pointer (Selects which VFD is used by EV-2)" %
%   N50:14/2  EV02_ENABLE_CR  "EV-2 Rotor Enable CR" %
%   N61:1  VFD_RUN_BITS_1  "These Bits Initcate the Status Off/Running for the appropriate VFD" %
%   N50:13/2  EV02_RUN  "EV-2 Rotor Running" %
% Rung: 4 %
% This Rung Starts EV-2 Rotor Drive
% when the operator presses the EV-2 PB
% AND
% the Interlocks are satisfied and the motor is Off %
SOR XIC N50:21/1 XIO N50:13/2 XIC N50:2/1 OTL N61:0/[N23:82] EOR
%   N50:21/1  EV02_PB_1S  "EV-2 Rotor Drive On/Off Pushbutton 1-Shot" %
%   N50:13/2  EV02_RUN  "EV-2 Rotor Running" %
%   N50:2/1  EV02_INTERLOCK  "EV-2 Rotor Drive Interlock 0 = Disable 1 = Enable" %
%   N61:0  VFD_ENABLE_BITS  "These Bits Enable the appropriate VFD" %
%   N23:82  EV02_OUT_PTR  "EV-2 Rotor Output Pointer (Selects which VFD is used by EV-2)" %
% Rung: 5 %
% his Rung Stops EV-2 Rotor Drive
% when the operator presses the EV-2 PB
% AND the motor is ON
% OR
% The Interlocks are NOT satisfied %
SOR BST XIC N50:21/1 XIC N50:13/2 NXB XIO N50:2/1 BND OTU N61:0/[N23:82] EOR
%   N50:21/1  EV02_PB_1S  "EV-2 Rotor Drive On/Off Pushbutton 1-Shot" %
%   N50:13/2  EV02_RUN  "EV-2 Rotor Running" %
%   N50:2/1  EV02_INTERLOCK  "EV-2 Rotor Drive Interlock 0 = Disable 1 = Enable" %
%   N61:0  VFD_ENABLE_BITS  "These Bits Enable the appropriate VFD" %
%   N23:82  EV02_OUT_PTR  "EV-2 Rotor Output Pointer (Selects which VFD is used by EV-2)" %

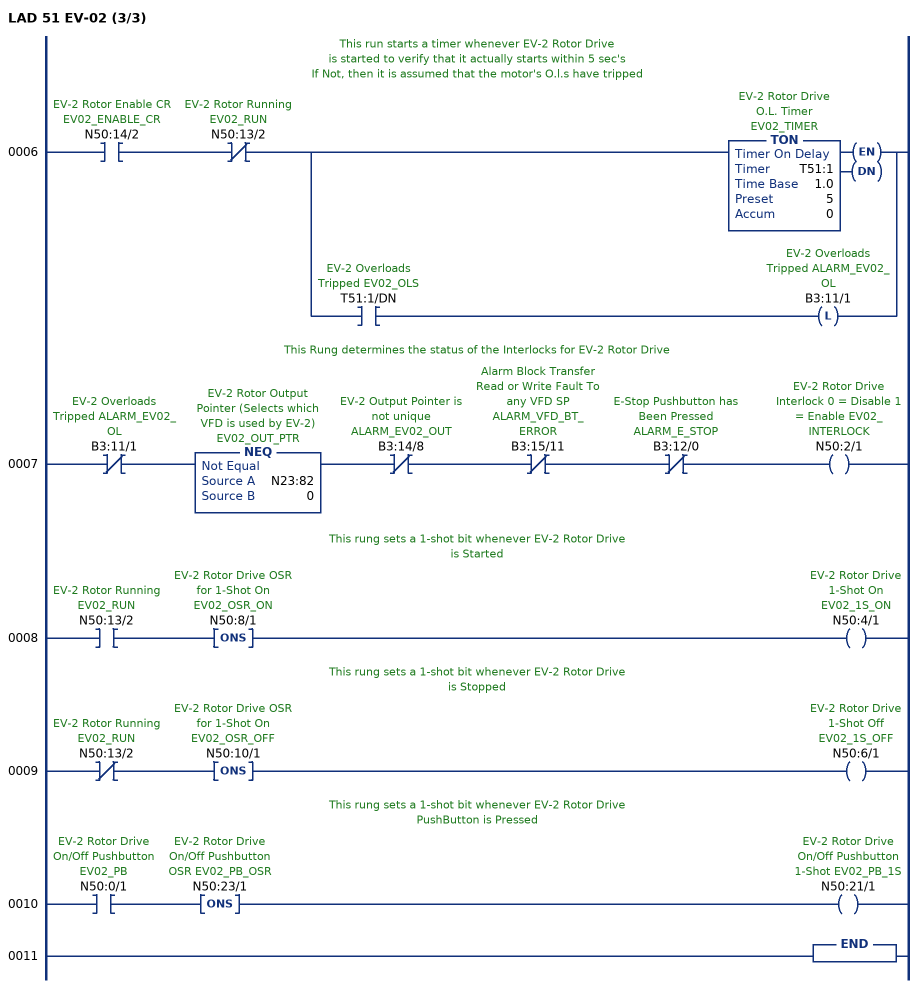
% Rung: 6 %
% This run starts a timer whenever EV-2 Rotor Drive
% is started to verify that it actually starts within 5 sec's
% If Not, then it is assumed that the motor's O.l.s have tripped %
SOR XIC N50:14/2 XIO N50:13/2 BST TON T51:1 1.0 5 0 NXB XIC T51:1/DN OTL B3:11/1 BND EOR
%   N50:14/2  EV02_ENABLE_CR  "EV-2 Rotor Enable CR" %
%   N50:13/2  EV02_RUN  "EV-2 Rotor Running" %
%   T51:1  EV02_TIMER  "EV-2 Rotor Drive O.L. Timer" %
%   T51:1/DN  EV02_OLS  "EV-2 Overloads Tripped" %
%   B3:11/1  ALARM_EV02_OL  "EV-2 Overloads Tripped" %
% Rung: 7 %
% This Rung determines the status of the Interlocks for EV-2 Rotor Drive %
SOR XIO B3:11/1 NEQ N23:82 0 XIO B3:14/8 XIO B3:15/11 XIO B3:12/0 OTE N50:2/1 EOR
%   B3:11/1  ALARM_EV02_OL  "EV-2 Overloads Tripped" %
%   N23:82  EV02_OUT_PTR  "EV-2 Rotor Output Pointer (Selects which VFD is used by EV-2)" %
%   B3:14/8  ALARM_EV02_OUT  "EV-2 Output Pointer is not unique" %
%   B3:15/11  ALARM_VFD_BT_ERROR  "Alarm Block Transfer Read or Write Fault To any VFD SP" %
%   B3:12/0  ALARM_E_STOP  "E-Stop Pushbutton has Been Pressed" %
%   N50:2/1  EV02_INTERLOCK  "EV-2 Rotor Drive Interlock 0 = Disable 1 = Enable" %
% Rung: 8 %
% This rung sets a 1-shot bit whenever EV-2 Rotor Drive
% is Started %
SOR XIC N50:13/2 OSR N50:8/1 OTE N50:4/1 EOR
%   N50:13/2  EV02_RUN  "EV-2 Rotor Running" %
%   N50:8/1  EV02_OSR_ON  "EV-2 Rotor Drive OSR for 1-Shot On" %
%   N50:4/1  EV02_1S_ON  "EV-2 Rotor Drive 1-Shot On" %
% Rung: 9 %
% This rung sets a 1-shot bit whenever EV-2 Rotor Drive
% is Stopped %
SOR XIO N50:13/2 OSR N50:10/1 OTE N50:6/1 EOR
%   N50:13/2  EV02_RUN  "EV-2 Rotor Running" %
%   N50:10/1  EV02_OSR_OFF  "EV-2 Rotor Drive OSR for 1-Shot On" %
%   N50:6/1  EV02_1S_OFF  "EV-2 Rotor Drive 1-Shot Off" %
% Rung: 10 %
% This rung sets a 1-shot bit whenever EV-2 Rotor Drive
% PushButton is Pressed %
SOR XIC N50:0/1 OSR N50:23/1 OTE N50:21/1 EOR
%   N50:0/1  EV02_PB  "EV-2 Rotor Drive On/Off Pushbutton" %
%   N50:23/1  EV02_PB_OSR  "EV-2 Rotor Drive On/Off Pushbutton OSR" %
%   N50:21/1  EV02_PB_1S  "EV-2 Rotor Drive On/Off Pushbutton 1-Shot" %
% Rung: 11 %
SOR END EOR

LADDER 52 "EV-03"    % EV-3 Rotor Drive VFD Controls %
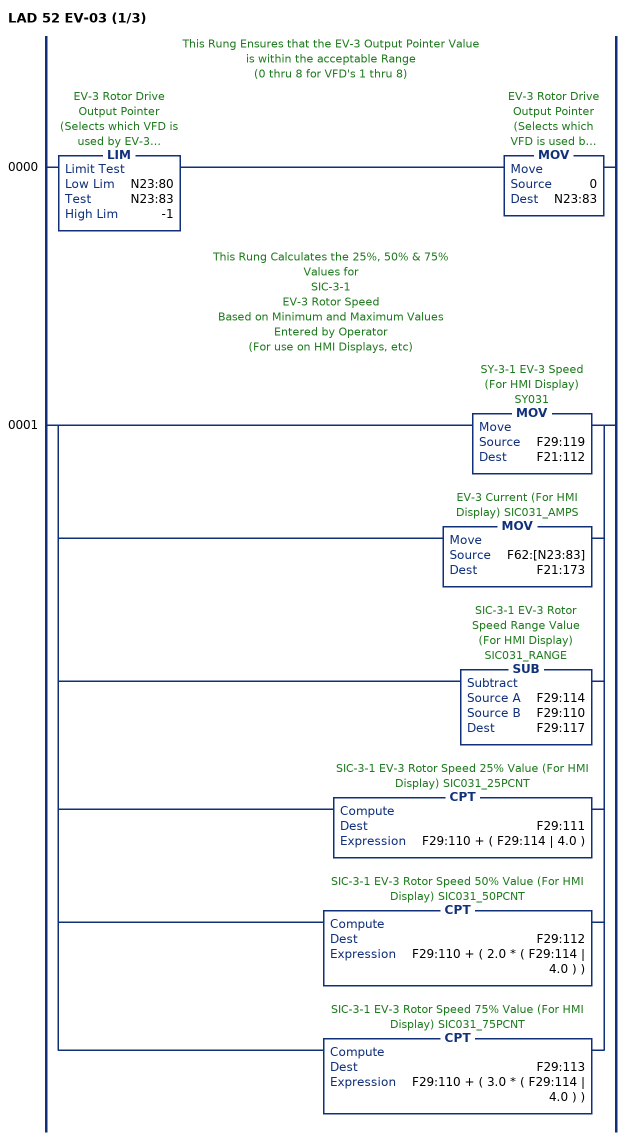
% Rung: 0 %
% This Rung Ensures that the EV-3 Output Pointer Value
% is within the acceptable Range
% (0 thru 8 for VFD's 1 thru 8) %
SOR LIM N23:80 N23:83 -1 MOV 0 N23:83 EOR
%   N23:80  MAX_VFD_ALLOWED_1  "Maximum Number of VFDs Available Plus 1" %
%   N23:83  EV03_OUT_PTR  "EV-3 Rotor Drive Output Pointer (Selects which VFD is used by EV-3)" %
% Rung: 1 %
% This Rung Calculates the 25%, 50% & 75%
% Values for
% SIC-3-1
% EV-3 Rotor Speed
% Based on Minimum and Maximum Values
% Entered by Operator
% (For use on HMI Displays, etc) %
SOR BST MOV F29:119 F21:112 NXB MOV F62:[N23:83] F21:173 NXB SUB F29:114 F29:110 F29:117 NXB CPT F29:111 " F29:110 + ( F29:114 | 4.0 ) " NXB CPT F29:112 " F29:110 + ( 2.0 * ( F29:114 | 4.0 ) ) " NXB CPT F29:113 " F29:110 + ( 3.0 * ( F29:114 | 4.0 ) ) " BND EOR
%   F29:119  SIC031_SP_FP  "SIC-3-1 EV-3 Rotor Speed Setpoint Value (For HMI Display)" %
%   F21:112  SY031  "SY-3-1 EV-3 Speed (For HMI Display)" %
%   N23:83  EV03_OUT_PTR  "EV-3 Rotor Drive Output Pointer (Selects which VFD is used by EV-3)" %
%   F21:173  SIC031_AMPS  "EV-3 Current (For HMI Display)" %
%   F29:114  SIC031_MAX  "SIC-3-1 EV-3 Rotor Speed 100% Value (For HMI Display)" %
%   F29:110  SIC031_MIN  "SIC-3-1 EV-3 Rotor Speed 0% Value (For HMI Display)" %
%   F29:117  SIC031_RANGE  "SIC-3-1 EV-3 Rotor Speed Range Value (For HMI Display)" %
%   F29:111  SIC031_25PCNT  "SIC-3-1 EV-3 Rotor Speed 25% Value (For HMI Display)" %
%   F29:112  SIC031_50PCNT  "SIC-3-1 EV-3 Rotor Speed 50% Value (For HMI Display)" %
%   F29:113  SIC031_75PCNT  "SIC-3-1 EV-3 Rotor Speed 75% Value (For HMI Display)" %

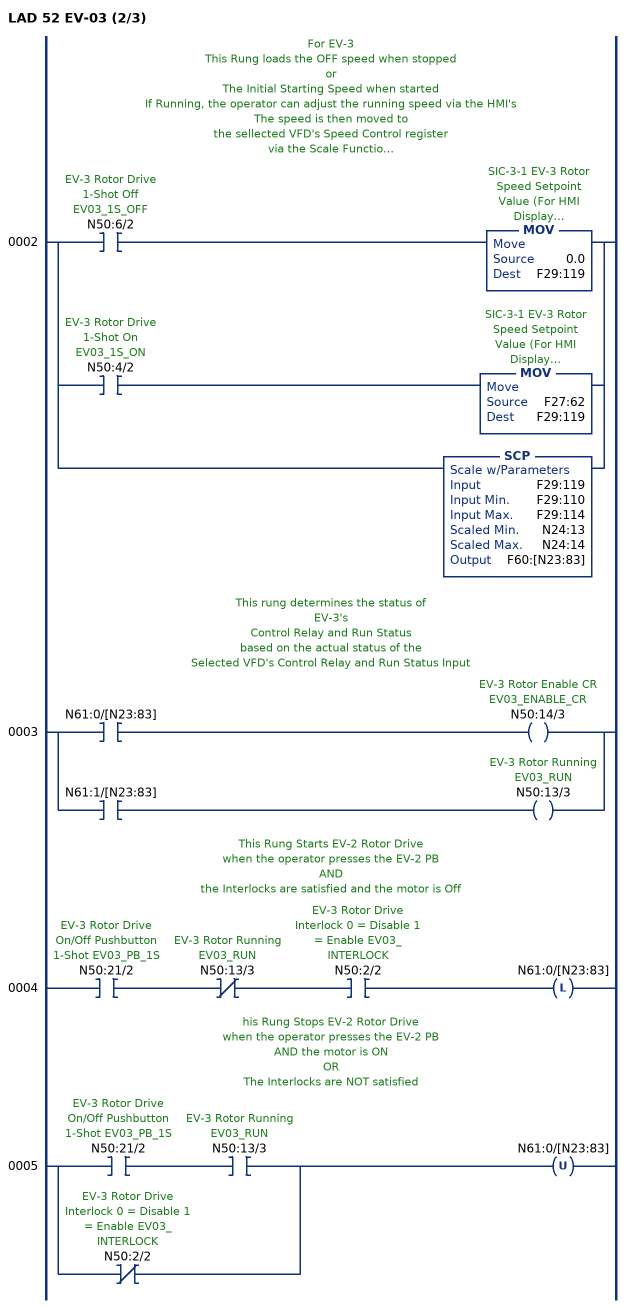
% Rung: 2 %
% For EV-3
% This Rung loads the OFF speed when stopped
% or
% The Initial Starting Speed when started
% If Running, the operator can adjust the running speed via the HMI's
% The speed is then moved to
% the sellected VFD's Speed Control register
% via the Scale Function
% to actually adjust the VFD's Speed %
SOR BST XIC N50:6/2 MOV 0.0 F29:119 NXB XIC N50:4/2 MOV F27:62 F29:119 NXB SCP F29:119 F29:110 F29:114 N24:13 N24:14 F60:[N23:83] BND EOR
%   N50:6/2  EV03_1S_OFF  "EV-3 Rotor Drive 1-Shot Off" %
%   F29:119  SIC031_SP_FP  "SIC-3-1 EV-3 Rotor Speed Setpoint Value (For HMI Display)" %
%   N50:4/2  EV03_1S_ON  "EV-3 Rotor Drive 1-Shot On" %
%   F27:62  SIC031_INIT_SP  "SY-3-1 Initial Speed Setpoint (RPM)" %
%   F29:110  SIC031_MIN  "SIC-3-1 EV-3 Rotor Speed 0% Value (For HMI Display)" %
%   F29:114  SIC031_MAX  "SIC-3-1 EV-3 Rotor Speed 100% Value (For HMI Display)" %
%   N24:13  AO_MIN_OE4  "Analog Output Minimum Value Generates 4 mA DC (To OE4 AO Module)" %
%   N24:14  AO_MAX_OE4  "Analog Output Maximum Value Generates 20 mA DC (To OE4 AO Module)" %
%   N23:83  EV03_OUT_PTR  "EV-3 Rotor Drive Output Pointer (Selects which VFD is used by EV-3)" %
% Rung: 3 %
% This rung determines the status of
% EV-3's
% Control Relay and Run Status
% based on the actual status of the
% Selected VFD's Control Relay and Run Status Input %
SOR BST XIC N61:0/[N23:83] OTE N50:14/3 NXB XIC N61:1/[N23:83] OTE N50:13/3 BND EOR
%   N61:0  VFD_ENABLE_BITS  "These Bits Enable the appropriate VFD" %
%   N23:83  EV03_OUT_PTR  "EV-3 Rotor Drive Output Pointer (Selects which VFD is used by EV-3)" %
%   N50:14/3  EV03_ENABLE_CR  "EV-3 Rotor Enable CR" %
%   N61:1  VFD_RUN_BITS_1  "These Bits Initcate the Status Off/Running for the appropriate VFD" %
%   N50:13/3  EV03_RUN  "EV-3 Rotor Running" %
% Rung: 4 %
% This Rung Starts EV-2 Rotor Drive
% when the operator presses the EV-2 PB
% AND
% the Interlocks are satisfied and the motor is Off %
SOR XIC N50:21/2 XIO N50:13/3 XIC N50:2/2 OTL N61:0/[N23:83] EOR
%   N50:21/2  EV03_PB_1S  "EV-3 Rotor Drive On/Off Pushbutton 1-Shot" %
%   N50:13/3  EV03_RUN  "EV-3 Rotor Running" %
%   N50:2/2  EV03_INTERLOCK  "EV-3 Rotor Drive Interlock 0 = Disable 1 = Enable" %
%   N61:0  VFD_ENABLE_BITS  "These Bits Enable the appropriate VFD" %
%   N23:83  EV03_OUT_PTR  "EV-3 Rotor Drive Output Pointer (Selects which VFD is used by EV-3)" %
% Rung: 5 %
% his Rung Stops EV-2 Rotor Drive
% when the operator presses the EV-2 PB
% AND the motor is ON
% OR
% The Interlocks are NOT satisfied %
SOR BST XIC N50:21/2 XIC N50:13/3 NXB XIO N50:2/2 BND OTU N61:0/[N23:83] EOR
%   N50:21/2  EV03_PB_1S  "EV-3 Rotor Drive On/Off Pushbutton 1-Shot" %
%   N50:13/3  EV03_RUN  "EV-3 Rotor Running" %
%   N50:2/2  EV03_INTERLOCK  "EV-3 Rotor Drive Interlock 0 = Disable 1 = Enable" %
%   N61:0  VFD_ENABLE_BITS  "These Bits Enable the appropriate VFD" %
%   N23:83  EV03_OUT_PTR  "EV-3 Rotor Drive Output Pointer (Selects which VFD is used by EV-3)" %

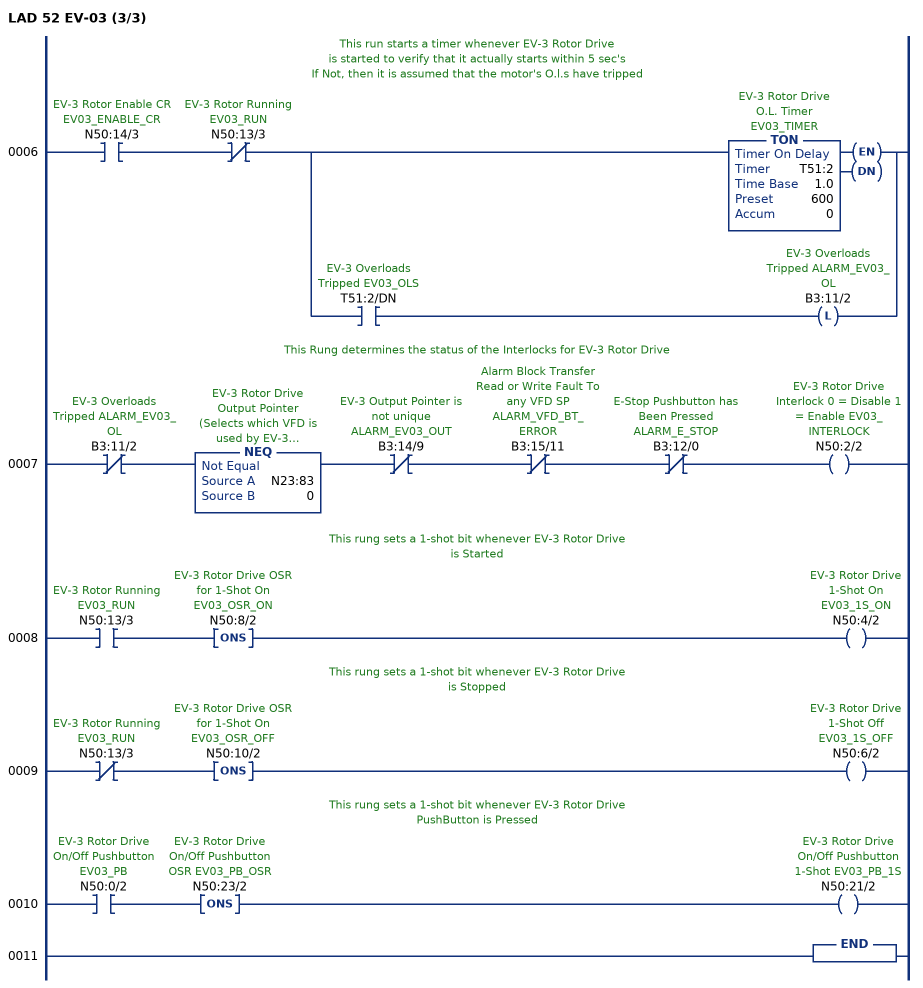
% Rung: 6 %
% This run starts a timer whenever EV-3 Rotor Drive
% is started to verify that it actually starts within 5 sec's
% If Not, then it is assumed that the motor's O.l.s have tripped %
SOR XIC N50:14/3 XIO N50:13/3 BST TON T51:2 1.0 600 0 NXB XIC T51:2/DN OTL B3:11/2 BND EOR
%   N50:14/3  EV03_ENABLE_CR  "EV-3 Rotor Enable CR" %
%   N50:13/3  EV03_RUN  "EV-3 Rotor Running" %
%   T51:2  EV03_TIMER  "EV-3 Rotor Drive O.L. Timer" %
%   T51:2/DN  EV03_OLS  "EV-3 Overloads Tripped" %
%   B3:11/2  ALARM_EV03_OL  "EV-3 Overloads Tripped" %
% Rung: 7 %
% This Rung determines the status of the Interlocks for EV-3 Rotor Drive %
SOR XIO B3:11/2 NEQ N23:83 0 XIO B3:14/9 XIO B3:15/11 XIO B3:12/0 OTE N50:2/2 EOR
%   B3:11/2  ALARM_EV03_OL  "EV-3 Overloads Tripped" %
%   N23:83  EV03_OUT_PTR  "EV-3 Rotor Drive Output Pointer (Selects which VFD is used by EV-3)" %
%   B3:14/9  ALARM_EV03_OUT  "EV-3 Output Pointer is not unique" %
%   B3:15/11  ALARM_VFD_BT_ERROR  "Alarm Block Transfer Read or Write Fault To any VFD SP" %
%   B3:12/0  ALARM_E_STOP  "E-Stop Pushbutton has Been Pressed" %
%   N50:2/2  EV03_INTERLOCK  "EV-3 Rotor Drive Interlock 0 = Disable 1 = Enable" %
% Rung: 8 %
% This rung sets a 1-shot bit whenever EV-3 Rotor Drive
% is Started %
SOR XIC N50:13/3 OSR N50:8/2 OTE N50:4/2 EOR
%   N50:13/3  EV03_RUN  "EV-3 Rotor Running" %
%   N50:8/2  EV03_OSR_ON  "EV-3 Rotor Drive OSR for 1-Shot On" %
%   N50:4/2  EV03_1S_ON  "EV-3 Rotor Drive 1-Shot On" %
% Rung: 9 %
% This rung sets a 1-shot bit whenever EV-3 Rotor Drive
% is Stopped %
SOR XIO N50:13/3 OSR N50:10/2 OTE N50:6/2 EOR
%   N50:13/3  EV03_RUN  "EV-3 Rotor Running" %
%   N50:10/2  EV03_OSR_OFF  "EV-3 Rotor Drive OSR for 1-Shot On" %
%   N50:6/2  EV03_1S_OFF  "EV-3 Rotor Drive 1-Shot Off" %
% Rung: 10 %
% This rung sets a 1-shot bit whenever EV-3 Rotor Drive
% PushButton is Pressed %
SOR XIC N50:0/2 OSR N50:23/2 OTE N50:21/2 EOR
%   N50:0/2  EV03_PB  "EV-3 Rotor Drive On/Off Pushbutton" %
%   N50:23/2  EV03_PB_OSR  "EV-3 Rotor Drive On/Off Pushbutton OSR" %
%   N50:21/2  EV03_PB_1S  "EV-3 Rotor Drive On/Off Pushbutton 1-Shot" %
% Rung: 11 %
SOR END EOR

LADDER 53 "AG-04"    % AG-4 Agitator Drive VFD Controls %
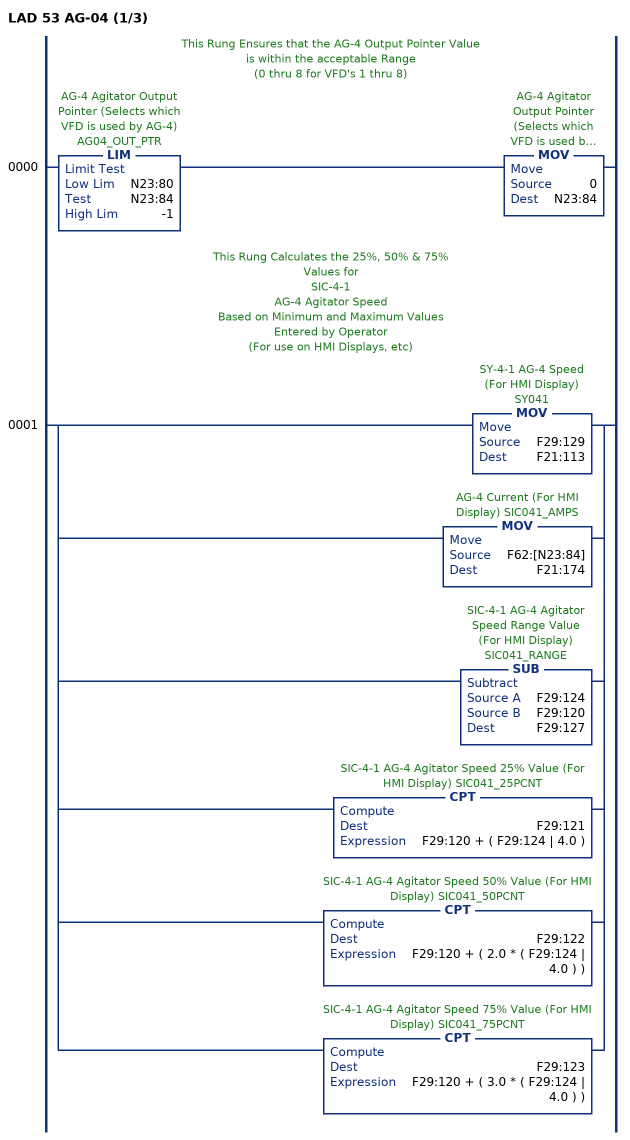
% Rung: 0 %
% This Rung Ensures that the AG-4 Output Pointer Value
% is within the acceptable Range
% (0 thru 8 for VFD's 1 thru 8) %
SOR LIM N23:80 N23:84 -1 MOV 0 N23:84 EOR
%   N23:80  MAX_VFD_ALLOWED_1  "Maximum Number of VFDs Available Plus 1" %
%   N23:84  AG04_OUT_PTR  "AG-4 Agitator Output Pointer (Selects which VFD is used by AG-4)" %
% Rung: 1 %
% This Rung Calculates the 25%, 50% & 75%
% Values for
% SIC-4-1
% AG-4 Agitator Speed
% Based on Minimum and Maximum Values
% Entered by Operator
% (For use on HMI Displays, etc) %
SOR BST MOV F29:129 F21:113 NXB MOV F62:[N23:84] F21:174 NXB SUB F29:124 F29:120 F29:127 NXB CPT F29:121 " F29:120 + ( F29:124 | 4.0 ) " NXB CPT F29:122 " F29:120 + ( 2.0 * ( F29:124 | 4.0 ) ) " NXB CPT F29:123 " F29:120 + ( 3.0 * ( F29:124 | 4.0 ) ) " BND EOR
%   F29:129  SIC041_SP_FP  "SIC-4-1 AG-4 Agitator Speed Setpoint Value (For HMI Display)" %
%   F21:113  SY041  "SY-4-1 AG-4 Speed (For HMI Display)" %
%   N23:84  AG04_OUT_PTR  "AG-4 Agitator Output Pointer (Selects which VFD is used by AG-4)" %
%   F21:174  SIC041_AMPS  "AG-4 Current (For HMI Display)" %
%   F29:124  SIC041_MAX  "SIC-4-1 AG-4 Agitator Speed 100% Value (For HMI Display)" %
%   F29:120  SIC041_MIN  "SIC-4-1 AG-4 Agitator Speed 0% Value (For HMI Display)" %
%   F29:127  SIC041_RANGE  "SIC-4-1 AG-4 Agitator Speed Range Value (For HMI Display)" %
%   F29:121  SIC041_25PCNT  "SIC-4-1 AG-4 Agitator Speed 25% Value (For HMI Display)" %
%   F29:122  SIC041_50PCNT  "SIC-4-1 AG-4 Agitator Speed 50% Value (For HMI Display)" %
%   F29:123  SIC041_75PCNT  "SIC-4-1 AG-4 Agitator Speed 75% Value (For HMI Display)" %

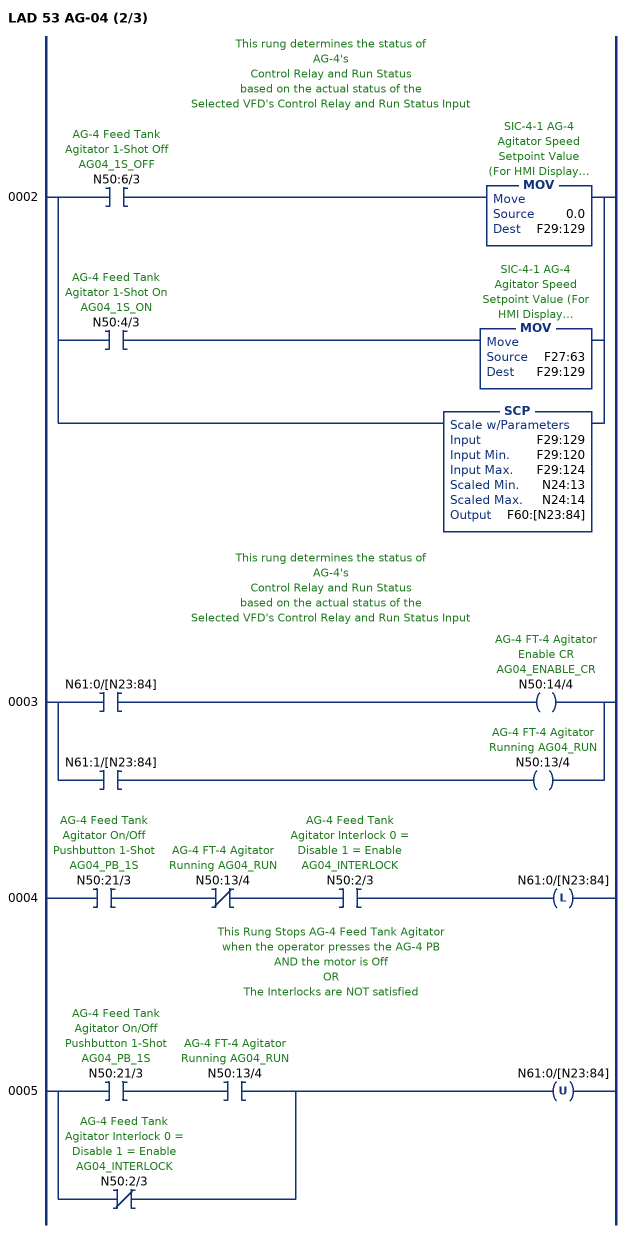
% Rung: 2 %
% This rung determines the status of
% AG-4's
% Control Relay and Run Status
% based on the actual status of the
% Selected VFD's Control Relay and Run Status Input %
SOR BST XIC N50:6/3 MOV 0.0 F29:129 NXB XIC N50:4/3 MOV F27:63 F29:129 NXB SCP F29:129 F29:120 F29:124 N24:13 N24:14 F60:[N23:84] BND EOR
%   N50:6/3  AG04_1S_OFF  "AG-4 Feed Tank Agitator 1-Shot Off" %
%   F29:129  SIC041_SP_FP  "SIC-4-1 AG-4 Agitator Speed Setpoint Value (For HMI Display)" %
%   N50:4/3  AG04_1S_ON  "AG-4 Feed Tank Agitator 1-Shot On" %
%   F27:63  SIC041_INIT_SP  "SY-4-1 Initial Speed Setpoint (RPM)" %
%   F29:120  SIC041_MIN  "SIC-4-1 AG-4 Agitator Speed 0% Value (For HMI Display)" %
%   F29:124  SIC041_MAX  "SIC-4-1 AG-4 Agitator Speed 100% Value (For HMI Display)" %
%   N24:13  AO_MIN_OE4  "Analog Output Minimum Value Generates 4 mA DC (To OE4 AO Module)" %
%   N24:14  AO_MAX_OE4  "Analog Output Maximum Value Generates 20 mA DC (To OE4 AO Module)" %
%   N23:84  AG04_OUT_PTR  "AG-4 Agitator Output Pointer (Selects which VFD is used by AG-4)" %
% Rung: 3 %
% This rung determines the status of
% AG-4's
% Control Relay and Run Status
% based on the actual status of the
% Selected VFD's Control Relay and Run Status Input %
SOR BST XIC N61:0/[N23:84] OTE N50:14/4 NXB XIC N61:1/[N23:84] OTE N50:13/4 BND EOR
%   N61:0  VFD_ENABLE_BITS  "These Bits Enable the appropriate VFD" %
%   N23:84  AG04_OUT_PTR  "AG-4 Agitator Output Pointer (Selects which VFD is used by AG-4)" %
%   N50:14/4  AG04_ENABLE_CR  "AG-4 FT-4 Agitator Enable CR" %
%   N61:1  VFD_RUN_BITS_1  "These Bits Initcate the Status Off/Running for the appropriate VFD" %
%   N50:13/4  AG04_RUN  "AG-4 FT-4 Agitator Running" %
% Rung: 4 %
SOR XIC N50:21/3 XIO N50:13/4 XIC N50:2/3 OTL N61:0/[N23:84] EOR
%   N50:21/3  AG04_PB_1S  "AG-4 Feed Tank Agitator On/Off Pushbutton 1-Shot" %
%   N50:13/4  AG04_RUN  "AG-4 FT-4 Agitator Running" %
%   N50:2/3  AG04_INTERLOCK  "AG-4 Feed Tank Agitator Interlock 0 = Disable 1 = Enable" %
%   N61:0  VFD_ENABLE_BITS  "These Bits Enable the appropriate VFD" %
%   N23:84  AG04_OUT_PTR  "AG-4 Agitator Output Pointer (Selects which VFD is used by AG-4)" %
% Rung: 5 %
% This Rung Stops AG-4 Feed Tank Agitator
% when the operator presses the AG-4 PB
% AND the motor is Off
% OR
% The Interlocks are NOT satisfied %
SOR BST XIC N50:21/3 XIC N50:13/4 NXB XIO N50:2/3 BND OTU N61:0/[N23:84] EOR
%   N50:21/3  AG04_PB_1S  "AG-4 Feed Tank Agitator On/Off Pushbutton 1-Shot" %
%   N50:13/4  AG04_RUN  "AG-4 FT-4 Agitator Running" %
%   N50:2/3  AG04_INTERLOCK  "AG-4 Feed Tank Agitator Interlock 0 = Disable 1 = Enable" %
%   N61:0  VFD_ENABLE_BITS  "These Bits Enable the appropriate VFD" %
%   N23:84  AG04_OUT_PTR  "AG-4 Agitator Output Pointer (Selects which VFD is used by AG-4)" %

